TYPE "PLC-Axis"	// UDT 31
VERSION : 0.0
  STRUCT
   A_FD_OR : BYTE ;	//Feedrate override
   A_DriveEnable : BOOL ;	//Drive test movement enable
   A_AckFixedStop : BOOL ;	//Acknowledge fixed stop reached
   A_SensorFixedStop : BOOL ;	//Sensor fixed stop
   A_ASpDisable : BOOL ;	//Axis/spindle disable
   A_Follow_upMode : BOOL ;	//Follow-up mode
   A_PosMeas1 : BOOL ;	//Position measuring system 1
   A_PosMeas2 : BOOL ;	//Position measuring system 2
   A_ORactive : BOOL ;	//Override active
   A_SWCam : BOOL ;	//SW cam activation
   A_ContrEnable : BOOL ;	//Controller enable
   A_DelDTGSpReset : BOOL ;	//Delete distance to go/Spindle-Reset
   A_Clamp : BOOL ;	//Clamping in progress
   A_RefVal1 : BOOL ;	//Reference point value 1
   A_RefVal2 : BOOL ;	//Reference point value 2
   A_RefVal3 : BOOL ;	//Reference point value 3
   A_RefVal4 : BOOL ;	//Reference point value 4
   A_ExtZO : BOOL ;	//Import external ZO
   A_EnabTravFixedStop : BOOL ;	//Enable travel to fixed stop
   A_FixedFD1 : BOOL ;	//Activate fixed feed 1
   A_FixedFD2 : BOOL ;	//Activate fixed feed 2
   A_FixedFD3 : BOOL ;	//Activate fixed feed 3
   A_FixedFD4 : BOOL ;	//Activate fixed feed 4
   A_VelocSpeedLimit : BOOL ;	//Velocity/spindle speed limitation
   A_PrgtestAxRel : BOOL ;	// Program test axis/spindle release
   A_HW1 : BOOL ;	//Activate handwheel 1
   A_HW2 : BOOL ;	//Activate handwheel 2
   A_HW3 : BOOL ;	//Activate handwheel 3
   A_FDSpStop : BOOL ;	//Feed stop/spindle stop
   A_Disable : BOOL ;	//Traversing key disable
   A_RapidTrOR : BOOL ;	//Rapid traverse override
   A_Minus : BOOL ;	//Traversing key minus
   A_Plus : BOOL ;	//Traversing key plus
   A_INC1 : BOOL ;	//INC1
   A_INC10 : BOOL ;	//INC10
   A_INC100 : BOOL ;	//INC100
   A_INC1000 : BOOL ;	//INC1000
   A_INC10000 : BOOL ;	//INC10000
   A_INCVar : BOOL ;	//INC variable
   A_OEMAxis : BYTE ;	//OEM axis signals
   A_InvHWDirOfRot : BOOL ;	// Inverting handwheel direction of rotation
   f7_1 : BOOL ;
   f7_2 : BOOL ;
   f7_3 : BOOL ;
   f7_4 : BOOL ;
   f7_5 : BOOL ;
   f7_6 : BOOL ;
   f7_7 : BOOL ;
   A_NCASpChanA : BOOL ;	//Assign NC axis/spindle channel A
   A_NCASpChanB : BOOL ;	//Assign NC axis/spindle channel B
   A_NCASpChanC : BOOL ;	//Assign NC axis/spindle channel C
   A_NCASpChanD : BOOL ;	//Assign NC axis/spindle channel D
   A_NCASpStrobe : BOOL ;	//Activation of assignment with pos. edge
   f8_5 : BOOL ;
   f8_6 : BOOL ;
   A_PLCASp : BOOL ;	//Request PLC axis/spindle
   A_Para_A : BOOL ;	//Parameter block servo A
   A_Para_B : BOOL ;	//Parameter block servo B
   A_Para_C : BOOL ;	//Parameter block servo C
   A_LockParSetDef : BOOL ;	//Lock parameter set definition from NC
   f9_4 : BOOL ;
   f9_5 : BOOL ;
   f9_6 : BOOL ;
   f9_7 : BOOL ;
   A_REPOSDelay : BOOL ;	//REPOS DELAY
   f10_1 : BOOL ;
   f10_2 : BOOL ;
   f10_3 : BOOL ;
   f10_4 : BOOL ;
   f10_5 : BOOL ;
   f10_6 : BOOL ;
   f10_7 : BOOL ;
   A_StartBrakeTest : BOOL ;	// Start brake test
   f11_1 : BOOL ;
   f11_2 : BOOL ;
   f11_3 : BOOL ;
   f11_4 : BOOL ;
   f11_5 : BOOL ;
   f11_6 : BOOL ;
   f11_7 : BOOL ;
   A_HWLimitMinus : BOOL ;	//Hardware limit switch minus
   A_HWLimitPlus : BOOL ;	//Hardware limit switch plus
   A_SWLimit2Minus : BOOL ;	//2nd software limit switch minus
   A_SWLimit2Plus : BOOL ;	//2nd software limit switch plus
   A_ModuloLimitEn : BOOL ;	// Modulo limit enabled
   f12_5 : BOOL ;
   f12_6 : BOOL ;
   A_DelayRef : BOOL ;	//Delay reference point approach
   A_JogFixPPos0 : BOOL ;	// JogFixPointPos 0
   A_JogFixPPos1 : BOOL ;	// JogFixPointPos 1
   A_JogFixPPos2 : BOOL ;	// JogFixPointPos 2
   A_JogToPos : BOOL ;	// Jog to position
   f13_4 : BOOL ;
   f13_5 : BOOL ;
   f13_6 : BOOL ;
   f13_7 : BOOL ;
   A_ProgtestSuppress : BOOL ;	// Program test to supress
   A_ProgtestActivate : BOOL ;	// Program test activate
   f14_2 : BOOL ;
   f14_3 : BOOL ;
   f14_4 : BOOL ;
   f14_5 : BOOL ;
   f14_6 : BOOL ;
   f14_7 : BOOL ;
   f15 : BYTE ;
   A_ActGearA : BOOL ;	//Actual gear stage A
   A_ActGearB : BOOL ;	//Actual gear stage B
   A_ActGearC : BOOL ;	//Actual gear stage C
   A_GearChangeOv : BOOL ;	//Gear has changed over
   A_Sp1Syn : BOOL ;	//Re-synchronize spindle 1
   A_Sp2Syn : BOOL ;	//Re-synchronize spindle 2
   A_NoMonitorGear : BOOL ;	//No monitoring when changing gear
   A_DeleteS : BOOL ;	//Delete S value
   A_FD_ORSp : BOOL ;	//Feedrate override for spindle valid
   f17_1 : BOOL ;
   f17_2 : BOOL ;
   f17_3 : BOOL ;
   A_Sp1SynP : BOOL ;	//Re-synchronize spindle 1 f. positioning
   A_Sp2SynP : BOOL ;	//Re-synchronize spindle 2 f. positioning
   A_M3M4Inv : BOOL ;	//Invert M3/M4
   f17_7 : BOOL ;
   f18_0 : BOOL ;
   f18_1 : BOOL ;
   f18_2 : BOOL ;
   f18_3 : BOOL ;
   A_OscilPLC : BOOL ;	//Oscillation via PLC
   A_OscilSpeed : BOOL ;	//enable Oscillation
   A_SetRotDirectRight : BOOL ;	//Setpoint osci. direct. right
   A_SetRotDirectLeft : BOOL ;	//Setpoint osci. direct. left
   A_SpOR : BYTE ;	//Spindle override
   f20_0 : BOOL ;
   A_RUEncQuStop : BOOL ;	//Run-up encoder quick stop
   f20_2 : BOOL ;
   A_SpeedSetpSmooth : BOOL ;	//Speed setpoint smoothing
   f20_4 : BOOL ;
   A_HoldBrakeToOpen : BOOL ;	// holding brake open
   f20_6 : BOOL ;
   f20_7 : BOOL ;
   A_ParA : BOOL ;	//Parameter set selection A
   A_ParB : BOOL ;	//Parameter set selection B
   A_ParC : BOOL ;	//Parameter set selection C
   A_MotA : BOOL ;	//Motor selection A
   A_MotB : BOOL ;	//Motor selection B
   A_MotOK : BOOL ;	//Motor selected
   A_IntegratDisable : BOOL ;	//n controller integrator disable
   A_PulseEnable : BOOL ;	//Pulse enable
   A_SG_SBH : BOOL ;	//Deselection SG/SBH
   A_SBH : BOOL ;	//Deselection of safe standstill
   f22_2 : BOOL ;
   A_SGselect0 : BOOL ;	//Selection SG bit 0
   A_SGselect1 : BOOL ;	//Selection SG bit 1
   f22_5 : BOOL ;
   f22_6 : BOOL ;
   f22_7 : BOOL ;
   A_Transmiss0 : BOOL ;	//Selection Transmission bit 0
   A_Transmiss1 : BOOL ;	//Selection Transmission bit 1
   A_Transmiss2 : BOOL ;	//Selection Transmission bit 2
   f23_3 : BOOL ;
   A_SE : BOOL ;	//Selection SE
   A_BrakeToClose : BOOL ;	//Sinamics: Brake to close
   f23_6 : BOOL ;
   A_TestStop : BOOL ;	//Activate test stop
   A_RotationMonit : BOOL ;	// Stepper motor: Rotation monitoring
   A_ControlAx : BOOL ;	// Control Axis
   f24_2 : BOOL ;
   f24_3 : BOOL ;
   A_TorqComp : BOOL ;	// Torque compensation
   A_ChangSetpOutAss0 : BOOL ;	// Bit value for CTRLOUT_changed - Change setpoint output assignment
   A_ChangSetpOutAss1 : BOOL ;	// Bit value for CTRLOUT_changed - Change setpoint output assignment
   A_MS : BOOL ;	//Master / Slave On
   f25 : BYTE ;
   f26_0 : BOOL ;
   f26_1 : BOOL ;
   f26_2 : BOOL ;
   A_CompContr : BOOL ;	//Compensation controller On
   A_FollowAxOv : BOOL ;	//Enable following axis override
   f26_5 : BOOL ;
   f26_6 : BOOL ;
   f26_7 : BOOL ;
   A_DEPMCS : BOOL ;	// Resume: DEPMCS
   A_DEPBCS : BOOL ;	// Resume: DEPBCS
   A_Corr : BOOL ;	// Resume: Corr
   A_HIAxMove : BOOL ;	// Resume: HIAxMove
   A_StopDEPMCS : BOOL ;	// Stop: DEPMCS
   A_StopDEPBCS : BOOL ;	// Stop: DEPBCS
   A_StopCorr : BOOL ;	// Stop: Corr
   A_StopHIAxMove : BOOL ;	// Stop: HIAxMove
   A_OscillAxExtRev : BOOL ;	// OscillAxExtReversal
   A_AxReset : BOOL ;	// AXRESET
   A_AxResume : BOOL ;	// AXRESUME
   A_SetRP : BOOL ;	//Set reversal point
   A_ChangeRP : BOOL ;	//Change reversal point
   A_StopRP : BOOL ;	//Stop at next reversal point
   A_Stop : BOOL ;	//Stop
   A_PLCAxis : BOOL ;	//PLC checks axis
   f29_0 : BOOL ;
   f29_1 : BOOL ;
   f29_2 : BOOL ;
   f29_3 : BOOL ;
   A_StartGantSynRun : BOOL ;	//Start gantry synchronization run
   A_NoAutoSync : BOOL ;	//No auto sync
   f29_6 : BOOL ;
   f29_7 : BOOL ;
   A_StopSpindle : BOOL ;	//Stop spindle
   A_StartCW : BOOL ;	//Start spindle Clockwise
   A_StartCCW : BOOL ;	//Start spindle Counterclockwise
   A_AutoGearStep : BOOL ;	//Autom. gear step change
   A_PosSpindle : BOOL ;	//Position spindle
   f30_5 : BOOL ;
   f30_6 : BOOL ;
   f30_7 : BOOL ;
   f31_0 : BOOL ;
   f31_1 : BOOL ;
   f31_2 : BOOL ;
   f31_3 : BOOL ;
   A_Resynchronize : BOOL ;	// Resynchronize
   A_DisSync : BOOL ;	// Disable synchronization
   A_Tracksync : BOOL ;	// Track synchronism
   A_DelSyncRunCorr : BOOL ;	// Deleting synchronous run correction
   f32_0 : BOOL ;
   f32_1 : BOOL ;
   A_extStopA : BOOL ;	//Deselection external Stop A
   A_extStopC : BOOL ;	//Deselection external Stop C
   A_extStopD : BOOL ;	//Deselection external Stop D
   A_extStopE : BOOL ;	//Deselection external Stop E
   f32_6 : BOOL ;
   f32_7 : BOOL ;
   f33_0 : BOOL ;
   f33_1 : BOOL ;
   f33_2 : BOOL ;
   f33_3 : BOOL ;
   A_SGcorr_0 : BOOL ;	//Selection SG-correction Bit 0
   A_SGcorr_1 : BOOL ;	//Selection SG-correction Bit 1
   A_SGcorr_2 : BOOL ;	//Selection SG-correction Bit 2
   A_SGcorr_3 : BOOL ;	//Selection SG-correction Bit 3
   f34 : ARRAY  [34 .. 55 ] OF BYTE ;
   A_FeedDriveCAxEng : BOOL ;	// Seperate feed drive as C axis engaged
   A_SpSpeedDisp : BOOL ;	// Spindle speed display
   A_SpInsideClamp : BOOL ;	// Spindle inside clamping
   f56_3 : BOOL ;
   f56_4 : BOOL ;
   f56_5 : BOOL ;
   f56_6 : BOOL ;
   f56_7 : BOOL ;
   f57 : BYTE ;
   f58 : WORD ;	// FC18: internal
   E_SpNA : BOOL ;	//Spindle/no axis
   E_NCU_Link : BOOL ;	//NCU_link active axis
   E_EncodFreq1 : BOOL ;	//Encoder limit frequency 1 exceeded
   E_EncodFreq2 : BOOL ;	//Encoder limit frequency 2 exceeded
   E_RefSyn1 : BOOL ;	//Referenced/synchronized 1
   E_RefSyn2 : BOOL ;	//Referenced/synchronized 2
   E_ExactCoarse : BOOL ;	//Position reached with exact stop coarse
   E_ExactFine : BOOL ;	//Position reached with exact stop fine
   E_TravRequ : BOOL ;	//Travel request
   E_AxialAlarm : BOOL ;	// Axial alarm
   E_AxisReady : BOOL ;	//Axis ready
   E_Follow_upMode : BOOL ;	//Follow-up mode active
   E_Stat : BOOL ;	//Axis/spindle stationary (n<nmin)
   E_PositContr : BOOL ;	//Position controller active
   E_SpeedContr : BOOL ;	//Speed controller active
   E_CurrentContr : BOOL ;	//Current controller active
   E_SWCam : BOOL ;	//Software cams active
   E_HWOverlay : BOOL ;	//Handwheel overlay active
   E_RevFD : BOOL ;	//Revolutional feedrate active
   E_MeasAct : BOOL ;	//Measuring active
   E_ActTravFStop : BOOL ;	//Activate travel to fixed stop
   E_FixedStop : BOOL ;	//Fixed stop reached
   E_ForceFixedStop : BOOL ;	// Force fixed stop limited
   E_AxContainerRot : BOOL ;	// Axis container rotation active
   E_AxReset : BOOL ;	// Axis reset done
   E_PLCCtrlAx : BOOL ;	// PLCcontrolled axis
   E_AxStop : BOOL ;	// Axis stop active
   E_AxSpDisable : BOOL ;	// Axis/spindle disable active
   E_StopDEPMCS : BOOL ;	// stop DEPMCS active
   E_StopDEPBCS : BOOL ;	// stop DEPBCS active
   E_StopCorr : BOOL ;	// stop Corr active
   E_StopHIAxMove : BOOL ;	// Stop HIAxMove active
   E_HW1 : BOOL ;	//Handwheel 1 active
   E_HW2 : BOOL ;	//Handwheel 2 active
   E_HW3 : BOOL ;	//Handwheel 3 active
   f64_3 : BOOL ;
   E_TReqMinus : BOOL ;	// Travel request minus
   E_TReqPlus : BOOL ;	// Travel request plus
   E_TCMinus : BOOL ;	//Traverse command minus
   E_TCPlus : BOOL ;	//Traverse command plus
   E_INC1 : BOOL ;	//INC1
   E_INC10 : BOOL ;	//INC10
   E_INC100 : BOOL ;	//INC100
   E_INC1000 : BOOL ;	//INC1000
   E_INC10000 : BOOL ;	//INC10000
   E_INCVar : BOOL ;	//INC variable
   f65_6 : BOOL ;
   f65_7 : BOOL ;
   E_OEMAxis : BYTE ;	//OEM axis signals
   E_InvHWDirOfRot : BOOL ;	// Handwheel direction of rotation invert actively
   f67_1 : BOOL ;
   f67_2 : BOOL ;
   f67_3 : BOOL ;
   f67_4 : BOOL ;
   f67_5 : BOOL ;
   f67_6 : BOOL ;
   f67_7 : BOOL ;
   E_NCASpChanA : BOOL ;	//NC axis/spindle in channel A
   E_NCASpChanB : BOOL ;	//NC axis/spindle in channel B
   E_NCASpChanC : BOOL ;	//NC axis/spindle in channel C
   E_NCASpChanD : BOOL ;	//NC axis/spindle in channel D
   E_PLCType : BOOL ;	//New type requested by PLC
   E_ChPoss : BOOL ;	//Change axis possible
   E_NeutrASp : BOOL ;	//Neutral axis/spindle
   E_PLCASp : BOOL ;	//PLC axis/spindle
   E_ParS_A : BOOL ;	//Parameter block servo A
   E_ParS_B : BOOL ;	//Parameter block servo B
   E_ParS_C : BOOL ;	//Parameter block servo C
   E_NCUNumLink_3 : BOOL ;
   E_NCUNumLink_4 : BOOL ;
   E_NCUNumLink_5 : BOOL ;
   E_NCUNumLink_6 : BOOL ;
   E_NCUNumLink_7 : BOOL ;
   E_ReposSh : BOOL ;	// Repos shift
   E_ReposShValid : BOOL ;	// Repos shift valid
   E_ReposDelayQuit : BOOL ;	// Repos delay quit
   f70_3 : BOOL ;
   f70_4 : BOOL ;
   f70_5 : BOOL ;
   f70_6 : BOOL ;
   f70_7 : BOOL ;
   E_BrakeTest : BOOL ;	// Brake test active
   f71_1 : BOOL ;
   f71_2 : BOOL ;
   f71_3 : BOOL ;
   E_POS_RESTORED1 : BOOL ;	// POS_RESTORED 1
   E_POS_RESTORED2 : BOOL ;	// POS_RESTORED 2
   f71_6 : BOOL ;
   E_PLCAxDedic : BOOL ;	// PLC Axis dedicated
   E_MMC_REPOSDelay : BOOL ;	//MMC REPOS DELAY
   f72_1 : BOOL ;
   f72_2 : BOOL ;
   f72_3 : BOOL ;
   f72_4 : BOOL ;
   f72_5 : BOOL ;
   f72_6 : BOOL ;
   f72_7 : BOOL ;
   f73 : BYTE ;
   f74_0 : BOOL ;
   f74_1 : BOOL ;
   f74_2 : BOOL ;
   f74_3 : BOOL ;
   E_ModLimEnAct : BOOL ;	// Modulo limit enabled active
   f74_5 : BOOL ;
   f74_6 : BOOL ;
   f74_7 : BOOL ;
   E_JogFixPPos0Act : BOOL ;	// JogFixPointPos 0 active
   E_JogFixPPos1Act : BOOL ;	// JogFixPointPos 1 active
   E_JogFixPPos2Act : BOOL ;	// JogFixPointPos 2 active
   E_JogFixPPos0 : BOOL ;	// JogFixPointPos 0 reached
   E_JogFixPPos1 : BOOL ;	// JogFixPointPos 1 reached
   E_JogFixPPos2 : BOOL ;	// JogFixPointPos 2 reached
   E_JogToPos : BOOL ;	// Jog to position active
   E_JogPos : BOOL ;	// Jog position reached
   E_ScratchPulse : BOOL ;	//Scratch pulse
   f76_1 : BOOL ;
   f76_2 : BOOL ;
   f76_3 : BOOL ;
   E_PathAxis : BOOL ;	// Path axis
   E_PosAxis : BOOL ;	//Positioning axis
   E_IndexAxisPos : BOOL ;	//Indexing axis in position
   E_CurvePos : BOOL ;	//Curve axis in position
   E_CollCheckRedSpeed : BOOL ;	//reduced speed of Collisions Check
   f77_1 : BOOL ;
   f77_2 : BOOL ;
   f77_3 : BOOL ;
   f77_4 : BOOL ;
   f77_5 : BOOL ;
   f77_6 : BOOL ;
   f77_7 : BOOL ;
   E_FPosAxis : REAL ;	//F function (REAL format) for positioning axes
   E_SetpGearA : BOOL ;	//Setpoint gear stage A
   E_SetpGearB : BOOL ;	//Setpoint gear stage B
   E_SetpGearC : BOOL ;	//Setpoint gear stage C
   E_GearChange : BOOL ;	//Gear changeover
   f82_4 : BOOL ;
   f82_5 : BOOL ;
   f82_6 : BOOL ;
   f82_7 : BOOL ;
   E_SpeedLimit : BOOL ;	//Speed limit exceeded
   E_SetSpeedLimit : BOOL ;	//Setpoint speed limited
   E_SetSpeedIncreased : BOOL ;	//Setpoint speed increased
   E_GeoMonit : BOOL ;	//Geometry monitoring
   E_SupportAreaViol : BOOL ;	//Support area limits violated
   E_SetRange : BOOL ;	//Spindle in setpoint range
   E_SpeedMonit : BOOL ;	//Speed monitoring
   E_ActRotRight : BOOL ;	//Actual rotation direction right
   E_ConstCuttSpeed : BOOL ;	//Const. cutting speed active
   E_SUG : BOOL ;	//SUG active (grinding wheel surface speed)
   E_CLG : BOOL ;	//CLG active
   E_Tapping : BOOL ;	//Tapping without compensating chuck
   E_SyncMode : BOOL ;	//Synchronous mode spindle active
   E_PosMode : BOOL ;	//Positioning mode spindle active
   E_OscillMode : BOOL ;	//Oscillation mode spindle active
   E_ContrMode : BOOL ;	//Control mode spindle active
   E_ToolDynLimit : BOOL ;	// Tool with limit of dynamics
   f85_1 : BOOL ;
   f85_2 : BOOL ;
   f85_3 : BOOL ;
   f85_4 : BOOL ;
   E_SpInPosition : BOOL ;	// Spindle in position
   f85_6 : BOOL ;
   f85_7 : BOOL ;
   E_MFunct : INT ;	//M function (INT) for spindle
   E_SFunct : REAL ;	//S function (REAL) for spindle
   f92_0 : BOOL ;
   E_RUEncDisabl : BOOL ;	//Run-up encoder disable active
   f92_2 : BOOL ;
   E_SpeedSetpSmooth : BOOL ;	//Speed setpoint smoothing active
   E_RLIact : BOOL ;	// RLI active
   E_HoldBrakeOpened : BOOL ;	// Holding brake opened
   f92_6 : BOOL ;
   f92_7 : BOOL ;
   E_ParA : BOOL ;	//Active parameter set A
   E_ParB : BOOL ;	//Active parameter set B
   E_ParC : BOOL ;	//Active parameter set C
   E_MotA : BOOL ;	//Active motor A
   E_MotB : BOOL ;	//Active motor B
   E_MotOK : BOOL ;	//Drive ready
   E_IntegratDisable : BOOL ;	//n controller integrator disabled
   E_PulseEnable : BOOL ;	//Pulses enabled
   E_MTempWarn : BOOL ;	//Temperature prewarning motor
   E_HTempWarn : BOOL ;	//Temperature prewarning heat sink
   E_RUComplete : BOOL ;	//Ramp-up complete
   E_MdMdx : BOOL ;	//Md<Mdx
   E_NactNmin : BOOL ;	//nact<nmin
   E_NactNx : BOOL ;	//nact<nx
   E_NactNset : BOOL ;	//nact<nset
   E_Message : BOOL ;	//Variable message function
   E_UDClessAlThreshold : BOOL ;	//UDC-link < alarm threshold
   f95_1 : BOOL ;
   f95_2 : BOOL ;
   f95_3 : BOOL ;
   f95_4 : BOOL ;
   f95_5 : BOOL ;
   f95_6 : BOOL ;
   f95_7 : BOOL ;	// Power Section I2T limit
   E_SpindleMonit : BOOL ;	//Error spindle monitoring
   E_AxisCtrl : BOOL ;	// Axis control active
   E_MSFine : BOOL ;	// Master/Slave fine
   E_MSCoarse : BOOL ;	// Master/Slave coarse
   E_MSCompContr : BOOL ;	// Master/Slave Compensation controller activ
   E_BitValCtrlOutChang0 : BOOL ;	// Bit value for CTRLOUT_changed 0:  Change setpoint output assignment
   E_BitValCtrlOutChang1 : BOOL ;	// Bit value for CTRLOUT_changed 1:  Change setpoint output assignment
   E_MS : BOOL ;	//Master/ slave active
   f97 : BYTE ;
   E_SyncronFine : BOOL ;	//Synchronism fine
   E_SyncronCoarse : BOOL ;	//Synchronism coarse
   E_ActValCoupling : BOOL ;	//Actual value coupling
   f98_3 : BOOL ;
   E_OverlayMotion : BOOL ;	//Overlaid motion
   E_SWL : BOOL ;	//Speed warning limit reached
   E_AWL : BOOL ;	//Acceleration warning limit reached
   E_EmRetr : BOOL ;	//Emergency retraction active
   E_MasterSp : BOOL ;	//Master spindle
   E_SlaveSp : BOOL ;	//Slave spindle
   E_SyncRunCorrDOut : BOOL ;	// Synchronous run correction driven out
   E_AxisAccel : BOOL ;	//Axis accelerated
   E_Sync : BOOL ;	//Synchronization active
   E_MSR : BOOL ;	//Max speed reached
   E_MAR : BOOL ;	//Max acceleration reached
   f99_7 : BOOL ;
   f100_0 : BOOL ;
   f100_1 : BOOL ;
   E_OscillAxExtRev : BOOL ;	// OscillAxExt Reversal active
   E_StopOscill : BOOL ;	//Oscillation cannot start
   E_ErrorOscill : BOOL ;	//Error during oscillation
   E_SparkOut : BOOL ;	//Spark-out active
   E_OscillMotion : BOOL ;	//Oscillation motion active
   E_Oscill : BOOL ;	//Oscillation active
   f101_0 : BOOL ;
   f101_1 : BOOL ;
   E_GantCOLimit : BOOL ;	//Gantry cut-off limit exceeded
   E_GantWarn : BOOL ;	//Gantry warning limit exceeded
   E_SynRunStart : BOOL ;	//Synchronization run ready to start
   E_GantGroupSyn : BOOL ;	//Gantry grouping is synchronous
   E_GantLeadAxis : BOOL ;	//Gantry leading axis
   E_GantAxis : BOOL ;	//Gantry axis
   f102 : BYTE ;
   E_SyncRunCorrIncl : BOOL ;	// Synchronous run correction is included
   f103_1 : BOOL ;
   f103_2 : BOOL ;
   f103_3 : BOOL ;
   f103_4 : BOOL ;
   f103_5 : BOOL ;
   f103_6 : BOOL ;
   f103_7 : BOOL ;
   E_AIAxis : ARRAY  [1 .. 31 ] OF BOOL ;	//Active infeed axis[1..31]
   E_SG_SBH : BOOL ;	//Active SG/SBH
   E_ErrLifeS_CRC : BOOL ;	// Error lifesign or CRC-error
   E_ImpdelNCK : BOOL ;	//Delete pulses NCK
   r108_3 : BOOL ;
   r108_4 : BOOL ;
   r108_5 : BOOL ;
   r108_6 : BOOL ;
   E_SRef : BOOL ;	//Axis safely referenced
   E_SN1Plus : BOOL ;	//Actual position > cam position SN1+
   E_SN1Minus : BOOL ;	//Actual position > cam position SN1-
   E_SN2Plus : BOOL ;	//Actual position > cam position SN2+
   E_SN2Minus : BOOL ;	//Actual position > cam position SN2-
   E_SN3Plus : BOOL ;	//Actual position > cam position SN3+
   E_SN3Minus : BOOL ;	//Actual position > cam position SN3-
   E_SN4Plus : BOOL ;	//Actual position > cam position SN4+
   E_SN4Minus : BOOL ;	//Actual position > cam position SN4-
   f110_0 : BOOL ;
   E_SBH : BOOL ;	//Active SBH
   f110_2 : BOOL ;
   E_SG_0 : BOOL ;	//Active SG 0
   E_SG_1 : BOOL ;	//Active SG 1
   E_n_nx : BOOL ;	//n < nx
   f110_6 : BOOL ;
   f110_7 : BOOL ;
   f111_0 : BOOL ;
   f111_1 : BOOL ;
   f111_2 : BOOL ;
   f111_3 : BOOL ;
   E_StopAB : BOOL ;	//Stop A/B active
   E_StopC : BOOL ;	//Stop C active
   E_StopD : BOOL ;	//Stop D active
   E_StopE : BOOL ;	//Stop E active
   E_CamRangeTr1 : BYTE ;	//Cam Range for Cam Track 1
   E_CamRangeTr2 : BYTE ;	//Cam Range for Cam Track 2
   E_CamRangeTr3 : BYTE ;	//Cam Range for Cam Track 3
   E_CamRangeTr4 : BYTE ;	//Cam Range for Cam Track 4
   f116 : BYTE ;
   E_CamTrack1 : BOOL ;	//Cam Track 1
   E_CamTrack2 : BOOL ;	//Cam Track 2
   E_CamTrack3 : BOOL ;	//Cam Track 3
   E_CamTrack4 : BOOL ;	//Cam Track 4
   f117_4 : BOOL ;
   f117_5 : BOOL ;
   f117_6 : BOOL ;
   f117_7 : BOOL ;
   E_CamRangeBitTr1 : ARRAY  [0 .. 14 ] OF //Cam Range Bits for Cam Track 1
   BOOL ;
   E_CamRangeBitTr2 : ARRAY  [0 .. 14 ] OF //Cam Range Bits for Cam Track 2
   BOOL ;
   E_CamRangeBitTr3 : ARRAY  [0 .. 14 ] OF //Cam Range Bits for Cam Track 3
   BOOL ;
   E_CamRangeBitTr4 : ARRAY  [0 .. 14 ] OF //Cam Range Bits for Cam Track 4
   BOOL ;
   f126 : WORD ;	// internal
   E_MMC_ProgtestSuppress : BOOL ;	// HMI->PLC: Program test to supress
   E_MMC_ProgtestActivate : BOOL ;	// HMI->PLC: Program test activate
   f128_2 : BOOL ;
   f128_3 : BOOL ;
   f128_4 : BOOL ;
   f128_5 : BOOL ;
   f128_6 : BOOL ;
   f128_7 : BOOL ;
   f129 : BYTE ;
   f130 : WORD ;
   E_SensorAv : BOOL ;	// Sensors available
   E_S1aMeasARod : BOOL ;	// Sensor S1: analogous measurement position of actuating rod
   f132_2 : BOOL ;
   f132_3 : BOOL ;
   E_S4dPistonStopP : BOOL ;	// Sensor S4: digital value piston stop position
   E_S5dAngleShaft : BOOL ;	// Sensor S5: digital value angle situation shaft
   f132_6 : BOOL ;
   f132_7 : BOOL ;
   f133 : BYTE ;
   E_ClampingState : INT ;	// state of the clamping system
   E_AnalogSensor : INT ;	// analog sensor on the motor
   f138_0 : BOOL ;
   f138_1 : BOOL ;
   f138_2 : BOOL ;
   f138_3 : BOOL ;
   E_S4PistonStopP : BOOL ;	// Sensor S4: piston stop position
   E_S5AngleShaft : BOOL ;	// Sensor S5: angle situation shaft
   f138_6 : BOOL ;
   f138_7 : BOOL ;
   f139 : BYTE ;
  END_STRUCT ;	
END_TYPE

// UDT 62: know-how protected block, not included

TYPE UDT 71
VERSION : 0.0
  STRUCT
   IFNo : ARRAY  [1 .. 16 ] OF BOOL ;	//Interface [no.] active
   Quit : ARRAY  [1 .. 16 ] OF BOOL ;	//perform Quit-End
   IF : ARRAY  [1 .. 16 ] OF STRUCT
    Loading : BOOL ;
    Unloading : BOOL ;
    Reloading : BOOL ;
    Positioning : BOOL ;
    PosbyProgram : BOOL ;	//Initiation by CNC Program
    PositioningMT : BOOL ;	//Positioning Multitool
    f0_6 : BOOL ;
    f0_7 : BOOL ;
    PerfStatusError : BOOL ;
    n1_1 : BOOL ;
    n1_2 : BOOL ;
    n1_3 : BOOL ;
    n1_4 : BOOL ;
    n1_5 : BOOL ;
    n1_6 : BOOL ;
    DataInDB1071 : BOOL ;
    Channel : BYTE ;	//Assigned channel
    TMno : BYTE ;	//Tool management no.
    Free1 : DINT ;	//Unassigned parameter 1
    Free2 : DINT ;	//Unassigned parameter 2
    Free3 : DINT ;	//Unassigned parameter 3
    IdentLoad : INT ;	//Identification for loading/unloading station
    NoLoad : INT ;	//No. of loading station
    SMag : INT ;	//Magazine no. (source) for unloading/reloading/pos.
    SLoc : INT ;	//Location no. (source) for unloading/reloading/pos.
    TMag : INT ;	//Magazine no. (target) for loading/reloading
    TLoc : INT ;	//Location no. (target) for loading/reloading
    WithoutMagMoving : BOOL ;	//HMI Data: Without Magazine Moving
    Res2 : BYTE ;
   END_STRUCT ;
  END_STRUCT ;	
END_TYPE

TYPE UDT 72
VERSION : 0.0
  STRUCT
   IFNo : ARRAY  [1 .. 16 ] OF BOOL ;	//Interface [no.] active
   Quit : ARRAY  [1 .. 16 ] OF BOOL ;	//perform Quit-End
   IF : ARRAY  [1 .. 16 ] OF STRUCT
    Comp : BOOL ;	//Compulsory change
    Perform : BOOL ;	//Perform change
    Prepare : BOOL ;	//Prepare change
    T0 : BOOL ;	//T0 programmed
    OldTinDBW42 : BOOL ;	//ZWS No. of Old Tool in DBW (n+42)
    ManTIn : BOOL ;	//Put in Tool in Spindle manual
    ManTOut : BOOL ;	//Get out Tool from Spindle manual
    SpiTRSpi : BOOL ;	//Spindle Tool remains in spindle
    PerfStatusError : BOOL ;
    n1_1 : BOOL ;
    n1_2 : BOOL ;
    n1_3 : BOOL ;
    n1_4 : BOOL ;
    n1_5 : BOOL ;
    n1_6 : BOOL ;
    DataInDB1072 : BOOL ;
    Channel : BYTE ;	//Assigned channel
    TMno : BYTE ;	//Tool management no.
    Free1 : DINT ;	//Unassigned parameter 1
    Free2 : DINT ;	//Unassigned parameter 2
    Free3 : DINT ;	//Unassigned parameter 3
    IdentBuff : INT ;	//Buffer identification (fixed value 9998)
    NoBuff : INT ;	//Relative location (target) in the buffer
    SMag : INT ;	//Magazine no. (source) for new tool
    SLoc : INT ;	//Location no. (source) for new tool
    TMag : INT ;	//Magazine no. (target) for old tool
    TLoc : INT ;	//Location no. (target) for old tool
    LocType : INT ;	//Tool new: location type
    SLeft : INT ;	//Tool new: size left
    SRight : INT ;	//Tool new: size right
    STop : INT ;	//Tool new: size top
    SBottom : INT ;	//Tool new: size bottom
    ToolInBuff : BOOL ;	//ID for tools in buffer
    IgnoreDisab : BOOL ;	//Ignore disabled
    TBUnloaded : BOOL ;	//To be unloaded
    TBLoaded : BOOL ;	//To be loaded
    MasterTool : BOOL ;	//Master tool
    n38_5 : BOOL ;	//reserved
    Exchange_1to1 : BOOL ;	//1:1 exchange
    HandTool : BOOL ;	//Hand tool
    ActTool : BOOL ;	//Active tool
    ToolEnabl : BOOL ;	//Tool enabled
    ToolDisab : BOOL ;	//Tool disabled
    Measured : BOOL ;	//Tool measured
    Prewarn : BOOL ;	//Prewarning limit reached
    ToolChange : BOOL ;	//Tool being changed
    FixedLoc : BOOL ;	//Tool fixed location coded
    ToolUsed : BOOL ;	//Tool was in use
    T_no : INT ;	//Tool new: T no.
    OldTZWSNo : INT ;	//ZWS No. of Old Tool
    MyMag : INT ;
    MyPlace : INT ;
   END_STRUCT ;
  END_STRUCT ;	
END_TYPE

TYPE UDT 73
VERSION : 0.0
  STRUCT
   IfNo : ARRAY  [1 .. 16 ] OF BOOL ;	//Interface [no.] active
   Quit : ARRAY  [1 .. 16 ] OF BOOL ;	//perform Quit-End
   IF : ARRAY  [1 .. 16 ] OF STRUCT
    Comp : BOOL ;	//Compulsory change
    Perform : BOOL ;	//Perform change
    f0_2 : BOOL ;
    T0 : BOOL ;	//T0 programmed
    f0_4 : BOOL ;
    f0_5 : BOOL ;
    ManTOut : BOOL ;	//Get out Tool from Holder manual
    f0_7 : BOOL ;
    PerfStatusError : BOOL ;
    n1_1 : BOOL ;
    n1_2 : BOOL ;
    n1_3 : BOOL ;
    n1_4 : BOOL ;
    n1_5 : BOOL ;
    n1_6 : BOOL ;
    DataInDB1073 : BOOL ;
    Channel : BYTE ;	//Assigned channel
    TMno : BYTE ;	//Tool management no.
    Free1 : DINT ;	//Unassigned parameter 1
    Free2 : DINT ;	//Unassigned parameter 2
    Free3 : DINT ;	//Unassigned parameter 3
    KennZWS : INT ;	//Reserved (buffer identification)
    NoBuff : INT ;	//Rel. location in buffer (res.)
    SMag : INT ;	//Magazine no. of turret
    SLoc : INT ;	//Location no. for new tool
    TMag : INT ;	//Magazine no. of turret (res.)
    TLoc : INT ;	//Location no. for old tool
    LocType : INT ;	//Tool new: location type
    SLeft : INT ;	//Tool new: size left
    SRight : INT ;	//Tool new: size right
    STop : INT ;	//Tool new: size top
    SBottom : INT ;	//Tool new: size bottom
    ToolInBuff : BOOL ;	//ID for tools in buffer
    IgnoreDisab : BOOL ;	//Ignore disabled
    TBUnloaded : BOOL ;	//To be unloaded
    TBLoaded : BOOL ;	//To be loaded
    MasterTool : BOOL ;	//Master tool
    n38_5 : BOOL ;	//reserved
    Exchange_1to1 : BOOL ;	//1:1 exchange
    HandTool : BOOL ;	//Hand tool
    ActTool : BOOL ;	//Active tool
    ToolEnabl : BOOL ;	//Tool enabled
    ToolDisab : BOOL ;	//Tool disabled
    Measured : BOOL ;	//Tool measured
    Prewarn : BOOL ;	//Prewarning limit reached
    ToolChange : BOOL ;	//Tool being changed
    FixedLoc : BOOL ;	//Tool fixed location coded
    ToolUsed : BOOL ;	//Tool was in use
    T_no : INT ;	//Tool new: T no.
    MyPlace : INT ;
   END_STRUCT ;
  END_STRUCT ;	
END_TYPE

TYPE UDT 77
VERSION : 0.0
  STRUCT
   MCP1In : ARRAY  [0 .. 7 ] OF BYTE ;
   MCP1Out : ARRAY  [0 .. 7 ] OF BYTE ;
   MCP1StatSend : DWORD ;
   MCP1StatRec : DWORD ;
   MCP2In : ARRAY  [0 .. 7 ] OF BYTE ;
   MCP2Out : ARRAY  [0 .. 7 ] OF BYTE ;
   MCP2StatSend : DWORD ;
   MCP2StatRec : DWORD ;
   BHGIn : ARRAY  [0 .. 5 ] OF BYTE ;
   Filler : ARRAY  [0 .. 5 ] OF BYTE ;
   BHGOut : ARRAY  [0 .. 19 ] OF BYTE ;
   BHGStatSend : DWORD ;
   BHGStatRec : DWORD ;
  END_STRUCT ;	
END_TYPE

TYPE UDT 1002
VERSION : 0.0
  STRUCT 	//Offset 0
   Chan : ARRAY  [1 .. 10 ] OF STRUCT 	//From Channel 1 to Channel 10
    FDD : ARRAY  [0 .. 15 ] OF //Feed disable
    BOOL ;
    RID : ARRAY  [0 .. 15 ] OF //Read-in disable
    BOOL ;
    NCSD : ARRAY  [0 .. 15 ] OF //NC start disable
    BOOL ;
    FdStop_1 : ARRAY  [0 .. 15 ] OF //Feed stop GEOaxis 1
    BOOL ;
    FdStop_2 : ARRAY  [0 .. 15 ] OF //Feed stop GEOaxis 2
    BOOL ;
    FdStop_3 : ARRAY  [0 .. 15 ] OF //Feed stop GEOaxis 3
    BOOL ;
   END_STRUCT ;	//without Alarmno for Chan (120 Byte)
//Offset 120
   Axis : ARRAY  [1 .. 31 ] OF STRUCT 	//From Axis 1 to Axis 31
    FdStop : ARRAY  [0 .. 15 ] OF //Feed stop axis/spindle 1
    BOOL ;
   END_STRUCT ;	//without Alarmno for Axis (62 Byte)
//Offset 182
   ZInfo0 : ARRAY  [0 .. 63 ] OF WORD ;	//Additional Value for UserAlarms 700000 to 700063
//Offset 310
   ChanA : ARRAY  [1 .. 10 ] OF STRUCT 	//From Channel 1 to Channel 10
    FDD_5C00xx : ARRAY  [0 .. 15 ] OF //Feed disable A.no.51000-510015
    BOOL ;
    FDD_RID_5C01xx : ARRAY  [0 .. 31 ] OF //Feed and read-in disable A.no.510100-510131
    BOOL ;
    RID_5C02xx : ARRAY  [0 .. 31 ] OF //Read-in disable A.no.510200-510231
    BOOL ;
    NCSD_5C03xx : ARRAY  [0 .. 15 ] OF //NC start disable A.no.510300-510315
    BOOL ;
    FdStop_1_5C11xx : ARRAY  [0 .. 15 ] OF //Feed stop GEOaxis 1 A.no.511100-511115
    BOOL ;
    FdStop_2_5C12xx : ARRAY  [0 .. 15 ] OF //Feed stop GEOaxis 2 A.no.511200-511215
    BOOL ;
    FdStop_3_5C13xx : ARRAY  [0 .. 15 ] OF //Feed stop GEOaxis 3 A.no.511300-511315
    BOOL ;
   END_STRUCT ;	//Alarmno for Chan are 5Cxxxx; C is the ChannelNo, except Channel 10. Channel 10
   AxisA : ARRAY  [1 .. 32 ] OF STRUCT 	//From Axis 1 to Axis 31
    AAFdStop60AAxx : ARRAY  [0 .. 15 ] OF //Feed stop axis/spindle
    BOOL ;
   END_STRUCT ;	//Alarmno for Axis are 60AAxx; A is the Axisno.
//Offset 554
   UserA : ARRAY  [0 .. 31 ] OF STRUCT
    A70UUxx : ARRAY  [0 .. 63 ] OF //Alarm 700000-700063 (user area 0)
    BOOL ;
   END_STRUCT ;	//Alarmno for UserAlarms are 7yUUxx; U is the Userarea, y = Db1004.UserDek2No[U]
  END_STRUCT ;	
END_TYPE

TYPE UDT 1071
VERSION : 0.0
  STRUCT
   MTIF : ARRAY  [1 .. 16 ] OF STRUCT
    MtType : INT ;
    MtPlaces : INT ;
    MtDistance : REAL ;
    MtNum : INT ;	// MT-No. to be positioned to
    MtPlaceNum : INT ;	// MT-PlaceNo. ~
    ToolHolder : INT ;	// TH-No as reference for MT-positioning
    IF : ARRAY  [1 .. 3 ] OF STRUCT
     reserved : INT ;	// reserved
    END_STRUCT ;
   END_STRUCT ;
  END_STRUCT ;	
END_TYPE

TYPE UDT 1072
VERSION : 0.0
  STRUCT
   MTIF : ARRAY  [1 .. 16 ] OF STRUCT
    MtType : INT ;
    MtPlaces : INT ;
    MtDistance : REAL ;
    MtNumNew : INT ;	// MT-No. new Tool
    MtPlaceNumNew : INT ;	// MtoolPlaceNum  ~
    MtNumOld : INT ;	// MT-No. old Tool
    MtPlaceNumOld : INT ;	// MtoolPlaceNum  ~
    LocType : INT ;	//Tool new: location type
    SLeft : INT ;	//Tool new: size left
    SRight : INT ;	//Tool new: size right
    STop : INT ;	//Tool new: size top
    SBottom : INT ;	//Tool new: size bottom
    ToolInBuff : BOOL ;	//ID for tools in buffer
    IgnoreDisab : BOOL ;	//Ignore disabled
    TBUnloaded : BOOL ;	//To be unloaded
    TBLoaded : BOOL ;	//To be loaded
    MasterTool : BOOL ;	//Master tool
    n26_5 : BOOL ;	//reserved
    n26_6 : BOOL ;	//reserved
    HandTool : BOOL ;	//Hand tool
    ActTool : BOOL ;	//Active tool
    ToolEnabl : BOOL ;	//Tool enabled
    ToolDisab : BOOL ;	//Tool disabled
    Measured : BOOL ;	//Tool measured
    Prewarn : BOOL ;	//Prewarning limit reached
    ToolChange : BOOL ;	//Tool being changed
    FixedLoc : BOOL ;	//Tool fixed location coded
    ToolUsed : BOOL ;	//Tool was in use
    T_no : INT ;	//Tool new: T no.
    ToolHolder : INT ;	// TH-No as tool compensation reference
    MtMyMag : INT ;	// MtoolNumber the tool is loaded onto
    MtMyPlace : INT ;	// MtoolPlaceNum ~
    IF : ARRAY  [1 .. 7 ] OF STRUCT
     reserved : INT ;	// reserved
    END_STRUCT ;
   END_STRUCT ;
  END_STRUCT ;	
END_TYPE

TYPE UDT 1073
VERSION : 0.0
  STRUCT
   MTIF : ARRAY  [1 .. 16 ] OF STRUCT
    MtType : INT ;
    MtPlaces : INT ;
    MtDistance : REAL ;
    MtNumNew : INT ;	// MT-No. new Tool
    MtPlaceNumNew : INT ;	// MtoolPlaceNum  ~
    MtNumOld : INT ;	// MT-No. old Tool
    MtPlaceNumOld : INT ;	// MtoolPlaceNum  ~
    LocType : INT ;	//Tool new: location type
    SLeft : INT ;	//Tool new: size left
    SRight : INT ;	//Tool new: size right
    STop : INT ;	//Tool new: size top
    SBottom : INT ;	//Tool new: size bottom
    ToolInBuff : BOOL ;	//ID for tools in buffer
    IgnoreDisab : BOOL ;	//Ignore disabled
    TBUnloaded : BOOL ;	//To be unloaded
    TBLoaded : BOOL ;	//To be loaded
    MasterTool : BOOL ;	//Master tool
    n26_5 : BOOL ;	//reserved
    n26_6 : BOOL ;	//reserved
    HandTool : BOOL ;	//Hand tool
    ActTool : BOOL ;	//Active tool
    ToolEnabl : BOOL ;	//Tool enabled
    ToolDisab : BOOL ;	//Tool disabled
    Measured : BOOL ;	//Tool measured
    Prewarn : BOOL ;	//Prewarning limit reached
    ToolChange : BOOL ;	//Tool being changed
    FixedLoc : BOOL ;	//Tool fixed location coded
    ToolUsed : BOOL ;	//Tool was in use
    T_no : INT ;	//Tool new: T no.
    ToolHolder : INT ;	// TH-No as tool compensation reference
    MtMyMag : INT ;	// MtoolNumber the tool is loaded onto
    MtMyPlace : INT ;	// MtoolPlaceNum ~
    IF : ARRAY  [1 .. 7 ] OF STRUCT
     reserved : INT ;	// reserved
    END_STRUCT ;
   END_STRUCT ;
  END_STRUCT ;	
END_TYPE

// FB 1: know-how protected block, not included

// FB 2: know-how protected block, not included

// FB 3: know-how protected block, not included

// FB 4: know-how protected block, not included

// FB 5: know-how protected block, not included

// FB 6: know-how protected block, not included

// FB 7: know-how protected block, not included

// FB 9: know-how protected block, not included

// FB 10: know-how protected block, not included

// FB 11: know-how protected block, not included

// FB 29: know-how protected block, not included

FUNCTION_BLOCK "Table_Ctrl"	// FB 100
AUTHOR : SEDIN
VERSION : 0.1
VAR
  Auxiliary : ARRAY  [0 .. 15 ] OF //Вспомогательная ячейка
  BOOL ;
END_VAR
VAR_TEMP
  ActMoment : INT ;	//Текущий момент, ось 1
END_VAR
BEGIN
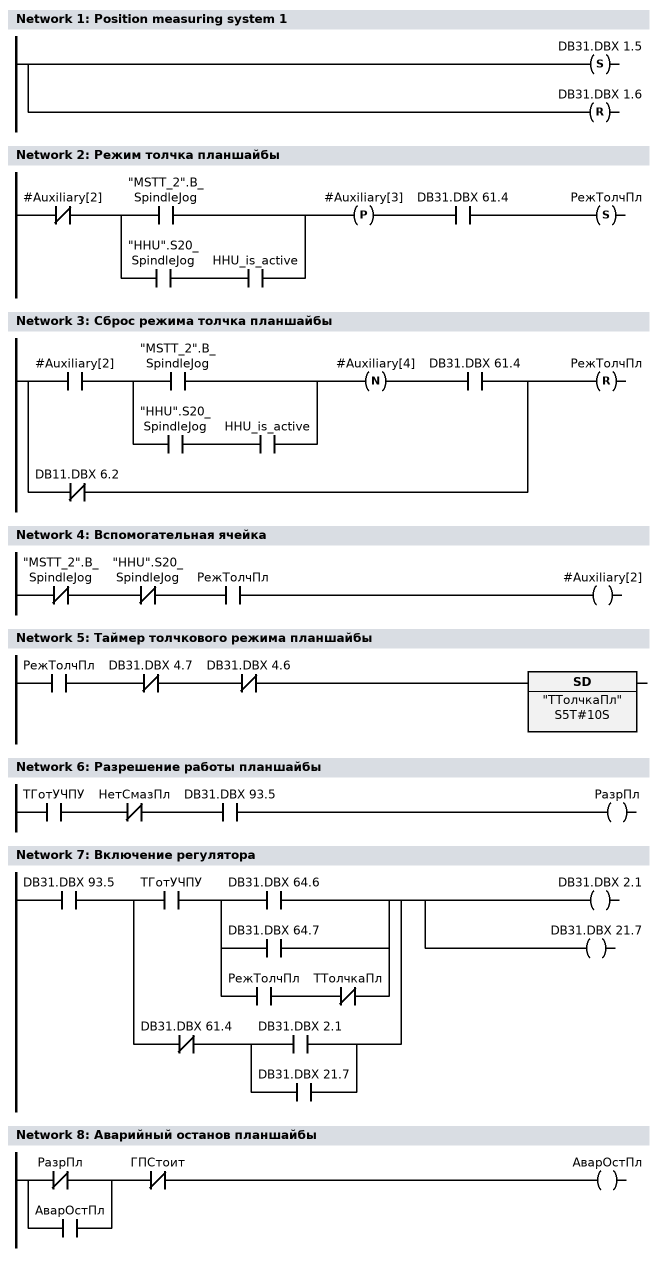
NETWORK
TITLE = Position measuring system 1
      SET;
      S     DB31.DBX 1.5;
      R     DB31.DBX 1.6;
NETWORK
TITLE = Режим толчка планшайбы
      AN    #Auxiliary[2];
      A(;
      O     "MSTT_2".B_SpindleJog;
      O;
      A     "HHU".S20_SpindleJog;
      A     "HHU_is_active";
      );
      FP    #Auxiliary[3];
      A     DB31.DBX 61.4;
      S     "РежТолчПл";
NETWORK
TITLE = Сброс режима толчка планшайбы
      A     #Auxiliary[2];
      A(;
      O     "MSTT_2".B_SpindleJog;
      O;
      A     "HHU".S20_SpindleJog;
      A     "HHU_is_active";
      );
      FN    #Auxiliary[4];
      A     DB31.DBX 61.4;
      ON    DB11.DBX 6.2;
      R     "РежТолчПл";
NETWORK
TITLE = Вспомогательная ячейка
      AN    "MSTT_2".B_SpindleJog;
      AN    "HHU".S20_SpindleJog;
      A     "РежТолчПл";
      =     #Auxiliary[2];
NETWORK
TITLE = Таймер толчкового режима планшайбы
      A     "РежТолчПл";
      AN    DB31.DBX 4.7;
      AN    DB31.DBX 4.6;
      L     S5T#10S;
      SD    "ТТолчкаПл";
NETWORK
TITLE = Разрешение работы планшайбы
      A     "ТГотУЧПУ";
      AN    "НетСмазПл";
      A     DB31.DBX 93.5;
      =     "РазрПл";
NETWORK
TITLE = Включение регулятора
      A     DB31.DBX 93.5;
      A(;
      A     "ТГотУЧПУ";
      A(;
      O     DB31.DBX 64.6;
      O     DB31.DBX 64.7;
      O;
      A     "РежТолчПл";
      AN    "ТТолчкаПл";
      );
      O;
      AN    DB31.DBX 61.4;
      A(;
      O     DB31.DBX 2.1;
      O     DB31.DBX 21.7;
      );
      );
      =     DB31.DBX 2.1;
      =     DB31.DBX 21.7;
NETWORK
TITLE = Аварийный останов планшайбы
      A(;
      ON    "РазрПл";
      O     "АварОстПл";
      );
      AN    "ГПСтоит";
      =     "АварОстПл";
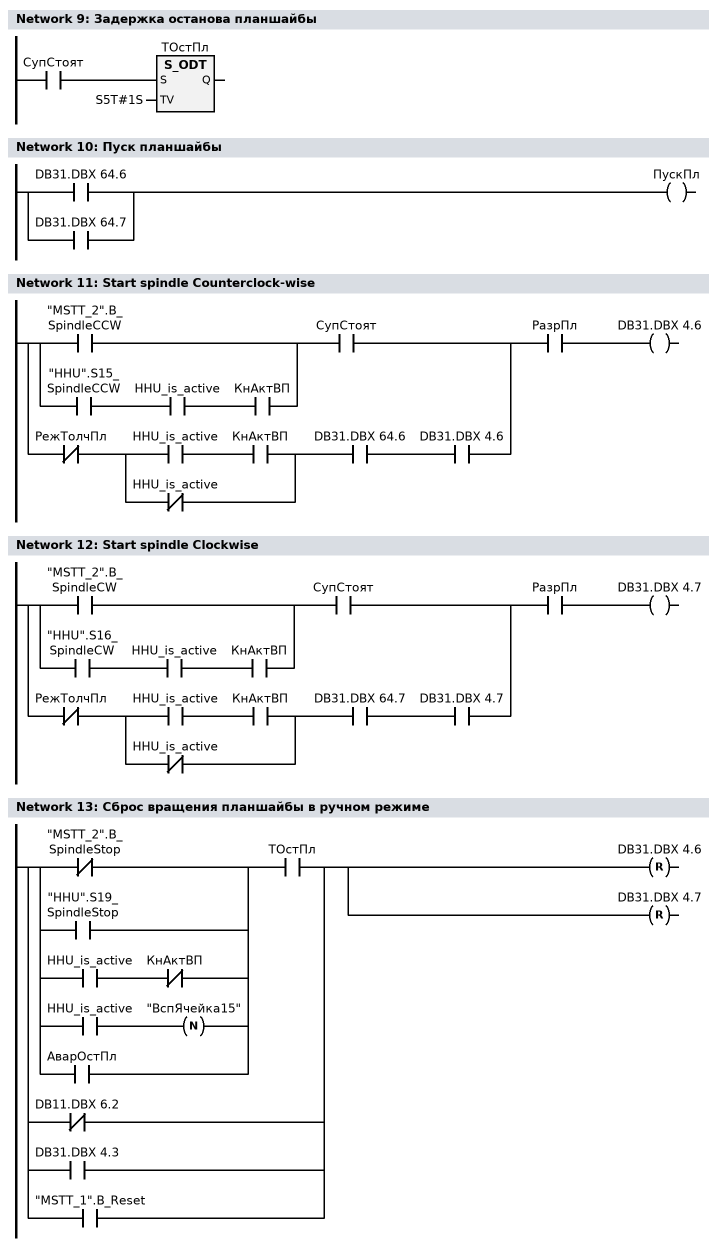
NETWORK
TITLE = Задержка останова планшайбы
      A     "СупСтоят";
      L     S5T#1S;
      SD    "ТОстПл";
      NOP   0;
      NOP   0;
      NOP   0;
      NOP   0;
NETWORK
TITLE = Пуск планшайбы
      O     DB31.DBX 64.6;
      O     DB31.DBX 64.7;
      =     "ПускПл";
NETWORK
TITLE = Start spindle Counterclock-wise
      A(;
      A(;
      O     "MSTT_2".B_SpindleCCW;
      O;
      A     "HHU".S15_SpindleCCW;
      A     "HHU_is_active";
      A     "КнАктВП";
      );
      A     "СупСтоят";
      O;
      AN    "РежТолчПл";
      A(;
      A     "HHU_is_active";
      A     "КнАктВП";
      ON    "HHU_is_active";
      );
      A     DB31.DBX 64.6;
      A     DB31.DBX 4.6;
      );
      A     "РазрПл";
      =     DB31.DBX 4.6;
NETWORK
TITLE = Start spindle Clockwise
      A(;
      A(;
      O     "MSTT_2".B_SpindleCW;
      O;
      A     "HHU".S16_SpindleCW;
      A     "HHU_is_active";
      A     "КнАктВП";
      );
      A     "СупСтоят";
      O;
      AN    "РежТолчПл";
      A(;
      A     "HHU_is_active";
      A     "КнАктВП";
      ON    "HHU_is_active";
      );
      A     DB31.DBX 64.7;
      A     DB31.DBX 4.7;
      );
      A     "РазрПл";
      =     DB31.DBX 4.7;
NETWORK
TITLE = Сброс вращения планшайбы в ручном режиме
      A(;
      ON    "MSTT_2".B_SpindleStop;
      O     "HHU".S19_SpindleStop;
      O(;
      A     "HHU_is_active";
      AN    "КнАктВП";
      );
      O(;
      A     "HHU_is_active";
      FN    "ВспЯчейка15";
      );
      O     "АварОстПл";
      );
      A     "ТОстПл";
      ON    DB11.DBX 6.2;
      O     DB31.DBX 4.3;
      O     "MSTT_1".B_Reset;
      R     DB31.DBX 4.6;
      R     DB31.DBX 4.7;
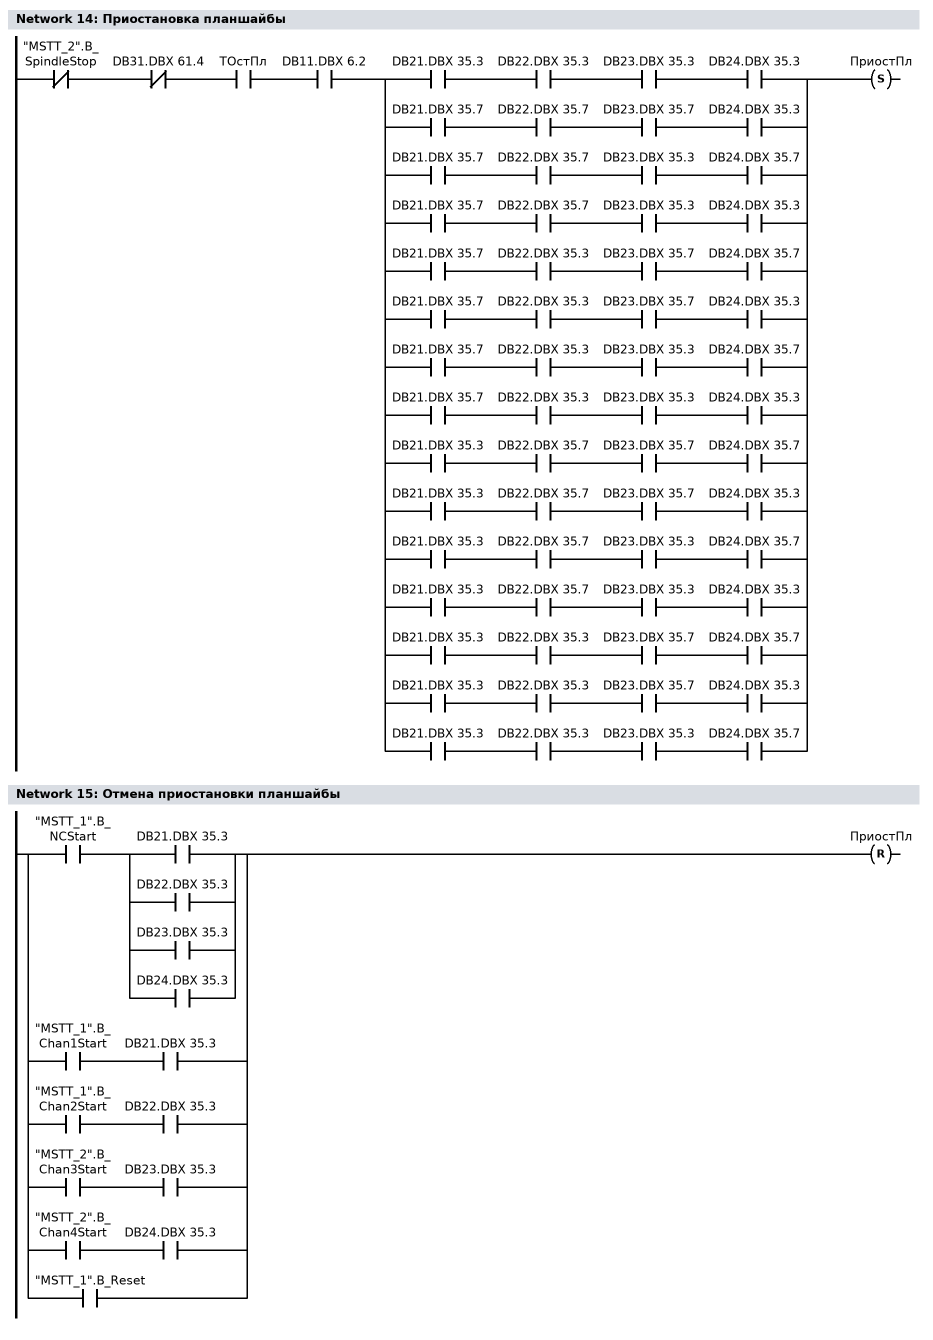
NETWORK
TITLE = Приостановка планшайбы
      AN    "MSTT_2".B_SpindleStop;
      AN    DB31.DBX 61.4;
      A     "ТОстПл";
      A     DB11.DBX 6.2;
      A(;
      A     DB21.DBX 35.3;
      A     DB22.DBX 35.3;
      A     DB23.DBX 35.3;
      A     DB24.DBX 35.3;
      O;
      A     DB21.DBX 35.7;
      A     DB22.DBX 35.7;
      A     DB23.DBX 35.7;
      A     DB24.DBX 35.3;
      O;
      A     DB21.DBX 35.7;
      A     DB22.DBX 35.7;
      A     DB23.DBX 35.3;
      A     DB24.DBX 35.7;
      O;
      A     DB21.DBX 35.7;
      A     DB22.DBX 35.7;
      A     DB23.DBX 35.3;
      A     DB24.DBX 35.3;
      O;
      A     DB21.DBX 35.7;
      A     DB22.DBX 35.3;
      A     DB23.DBX 35.7;
      A     DB24.DBX 35.7;
      O;
      A     DB21.DBX 35.7;
      A     DB22.DBX 35.3;
      A     DB23.DBX 35.7;
      A     DB24.DBX 35.3;
      O;
      A     DB21.DBX 35.7;
      A     DB22.DBX 35.3;
      A     DB23.DBX 35.3;
      A     DB24.DBX 35.7;
      O;
      A     DB21.DBX 35.7;
      A     DB22.DBX 35.3;
      A     DB23.DBX 35.3;
      A     DB24.DBX 35.3;
      O;
      A     DB21.DBX 35.3;
      A     DB22.DBX 35.7;
      A     DB23.DBX 35.7;
      A     DB24.DBX 35.7;
      O;
      A     DB21.DBX 35.3;
      A     DB22.DBX 35.7;
      A     DB23.DBX 35.7;
      A     DB24.DBX 35.3;
      O;
      A     DB21.DBX 35.3;
      A     DB22.DBX 35.7;
      A     DB23.DBX 35.3;
      A     DB24.DBX 35.7;
      O;
      A     DB21.DBX 35.3;
      A     DB22.DBX 35.7;
      A     DB23.DBX 35.3;
      A     DB24.DBX 35.3;
      O;
      A     DB21.DBX 35.3;
      A     DB22.DBX 35.3;
      A     DB23.DBX 35.7;
      A     DB24.DBX 35.7;
      O;
      A     DB21.DBX 35.3;
      A     DB22.DBX 35.3;
      A     DB23.DBX 35.7;
      A     DB24.DBX 35.3;
      O;
      A     DB21.DBX 35.3;
      A     DB22.DBX 35.3;
      A     DB23.DBX 35.3;
      A     DB24.DBX 35.7;
      );
      S     "ПриостПл";
NETWORK
TITLE = Отмена приостановки планшайбы
      A     "MSTT_1".B_NCStart;
      A(;
      O     DB21.DBX 35.3;
      O     DB22.DBX 35.3;
      O     DB23.DBX 35.3;
      O     DB24.DBX 35.3;
      );
      O;
      A     "MSTT_1".B_Chan1Start;
      A     DB21.DBX 35.3;
      O;
      A     "MSTT_1".B_Chan2Start;
      A     DB22.DBX 35.3;
      O;
      A     "MSTT_2".B_Chan3Start;
      A     DB23.DBX 35.3;
      O;
      A     "MSTT_2".B_Chan4Start;
      A     DB24.DBX 35.3;
      O     "MSTT_1".B_Reset;
      R     "ПриостПл";
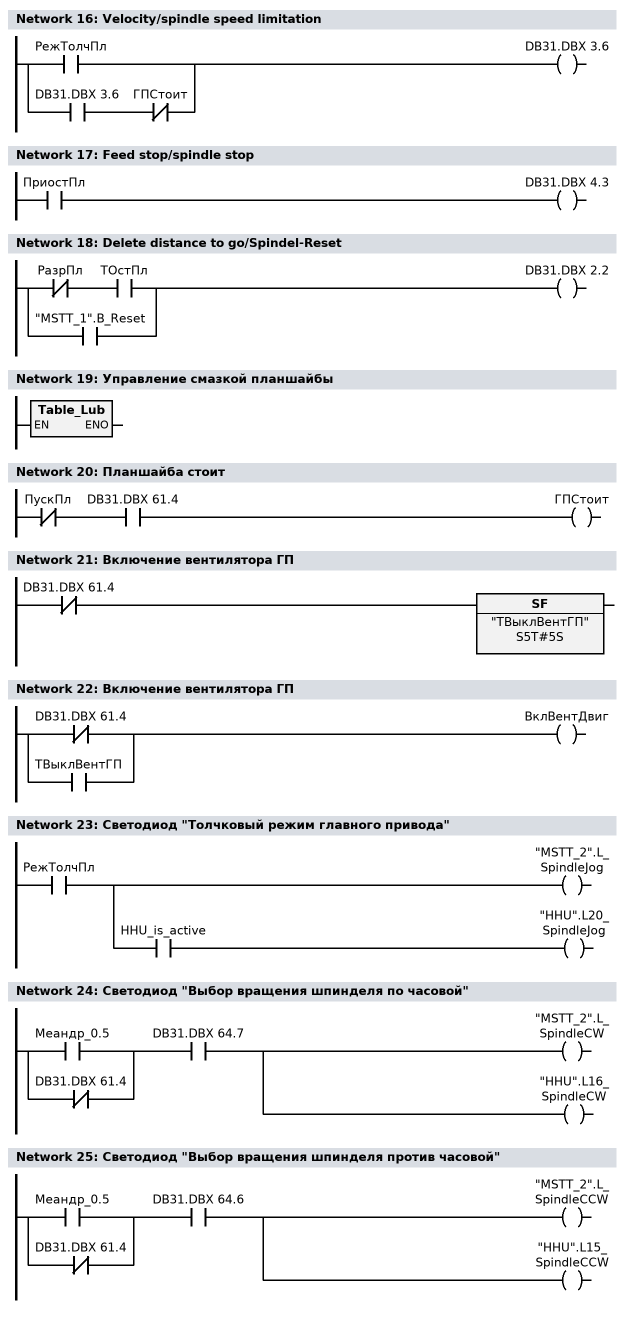
NETWORK
TITLE = Velocity/spindle speed limitation
      O     "РежТолчПл";
      O;
      A     DB31.DBX 3.6;
      AN    "ГПСтоит";
      =     DB31.DBX 3.6;
NETWORK
TITLE = Feed stop/spindle stop
      A     "ПриостПл";
      =     DB31.DBX 4.3;
NETWORK
TITLE = Delete distance to go/Spindel-Reset
      AN    "РазрПл";
      A     "ТОстПл";
      O     "MSTT_1".B_Reset;
      =     DB31.DBX 2.2;
NETWORK
TITLE = Управление смазкой планшайбы
      CALL  "Table_Lub";
      NOP   0;
NETWORK
TITLE = Планшайба стоит
      AN    "ПускПл";
      A     DB31.DBX 61.4;
      =     "ГПСтоит";
NETWORK
TITLE = Включение вентилятора ГП
      AN    DB31.DBX 61.4;
      L     S5T#5S;
      SF    "ТВыклВентГП";
NETWORK
TITLE = Включение вентилятора ГП
      ON    DB31.DBX 61.4;
      O     "ТВыклВентГП";
      =     "ВклВентДвиг";
NETWORK
TITLE = Светодиод "Толчковый режим главного привода"
      A     "РежТолчПл";
      =     L 2.0;
      A     L 2.0;
      BLD   102;
      =     "MSTT_2".L_SpindleJog;
      A     L 2.0;
      A     "HHU_is_active";
      =     "HHU".L20_SpindleJog;
NETWORK
TITLE = Светодиод "Выбор вращения шпинделя по часовой"
      A(;
      O     "Меандр_0.5";
      ON    DB31.DBX 61.4;
      );
      A     DB31.DBX 64.7;
      =     "MSTT_2".L_SpindleCW;
      =     "HHU".L16_SpindleCW;
NETWORK
TITLE = Светодиод "Выбор вращения шпинделя против часовой"
      A(;
      O     "Меандр_0.5";
      ON    DB31.DBX 61.4;
      );
      A     DB31.DBX 64.6;
      =     "MSTT_2".L_SpindleCCW;
      =     "HHU".L15_SpindleCCW;
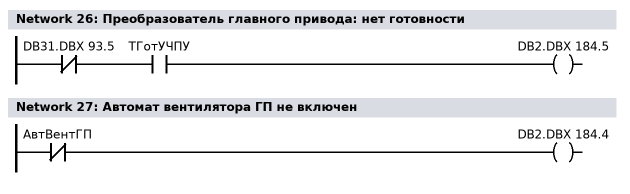
NETWORK
TITLE = Преобразователь главного привода: нет готовности
      AN    DB31.DBX 93.5;
      A     "ТГотУЧПУ";
      =     DB2.DBX 184.5;
NETWORK
TITLE = Автомат вентилятора ГП не включен
      AN    "АвтВентГП";
      =     DB2.DBX 184.4;
END_FUNCTION_BLOCK

FUNCTION_BLOCK "Support1_Ctrl"	// FB 101
AUTHOR : SEDIN
VERSION : 0.1
VAR
  Auxiliary : ARRAY  [0 .. 15 ] OF //Вспомогательная ячейка
  BOOL ;
  Unbrake1 : BOOL ;	//Требование разжима оси 1
  Unbrake2 : BOOL ;	//Требование разжима оси 2
  ErrorLub : BOOL ;	//Ошибка ИСС
  Sup_Lub : FB 121;	//Управление смазкой суппорта
  StartFC18_1 : BOOL ;	//Старт FC18
  StopFC18_1 : BOOL ;	//Остановка FC18
  InPosFC18_1 : BOOL ;	//Выполнение FC18
  ErrorFC18_1 : BOOL ;	//Ошибка FC18
  StartFC18_2 : BOOL ;	//Старт FC18
  StopFC18_2 : BOOL ;	//Остановка FC18
  InPosFC18_2 : BOOL ;	//Выполнение FC18
  ErrorFC18_2 : BOOL ;	//Ошибка FC18
  StateFC18_1 : BYTE ;	//Состояние FC18
  StateFC18_2 : BYTE ;	//Состояние FC18
END_VAR
VAR_TEMP
  Permission : BOOL ;	//Разрешение работы суппорта
  Permission1 : BOOL ;	//Разрешение работы суппорта, ось 1
  Permission2 : BOOL ;	//Разрешение работы суппорта, ось 2
  JogStop : BOOL ;	//Останов подачи в ручном режиме
  Stop1 : BOOL ;	//Суппорт стоит, ось 1
  Stop2 : BOOL ;	//Суппорт стоит, ось 2
  ErrorLub1 : BOOL ;	//Низкий уровень масла в ИСС
  ErrorLub2 : BOOL ;	//Не достигнуто давление в ИСС
  ErrorLub3 : BOOL ;	//Нет падения давления в ИСС
END_VAR
BEGIN
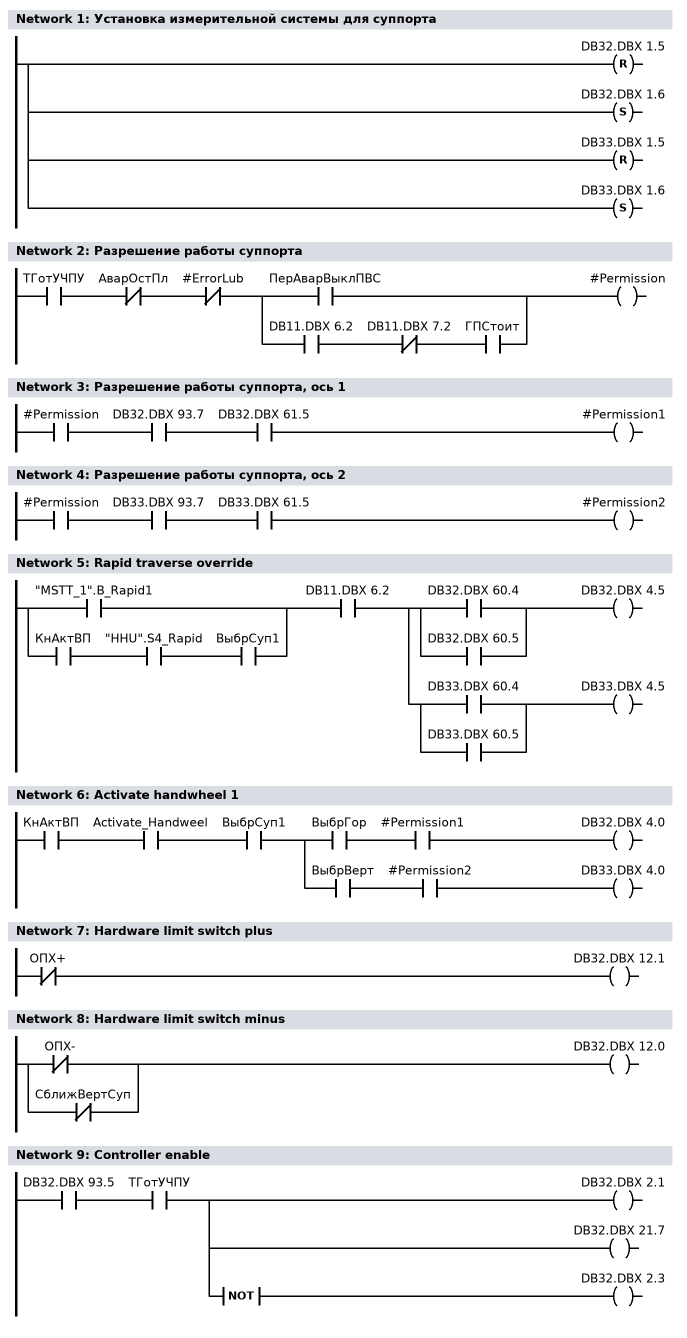
NETWORK
TITLE = Установка измерительной системы для суппорта
      SET;
      R     DB32.DBX 1.5;
      S     DB32.DBX 1.6;
      R     DB33.DBX 1.5;
      S     DB33.DBX 1.6;
NETWORK
TITLE = Разрешение работы суппорта
      A     "ТГотУЧПУ";
      AN    "АварОстПл";
      AN    #ErrorLub;
      A(;
      O     "ПерАварВыклПВС";
      O;
      A     DB11.DBX 6.2;
      AN    DB11.DBX 7.2;
      A     "ГПСтоит";
      );
      =     #Permission;
NETWORK
TITLE = Разрешение работы суппорта, ось 1
      A     #Permission;
      A     DB32.DBX 93.7;
      A     DB32.DBX 61.5;
      =     #Permission1;
NETWORK
TITLE = Разрешение работы суппорта, ось 2
      A     #Permission;
      A     DB33.DBX 93.7;
      A     DB33.DBX 61.5;
      =     #Permission2;
NETWORK
TITLE = Rapid traverse override
      A(;
      O     "MSTT_1".B_Rapid1;
      O;
      A     "КнАктВП";
      A     "HHU".S4_Rapid;
      A     "ВыбрСуп1";
      );
      A     DB11.DBX 6.2;
      =     L 2.0;
      A     L 2.0;
      A(;
      O     DB32.DBX 60.4;
      O     DB32.DBX 60.5;
      );
      =     DB32.DBX 4.5;
      A     L 2.0;
      A(;
      O     DB33.DBX 60.4;
      O     DB33.DBX 60.5;
      );
      =     DB33.DBX 4.5;
NETWORK
TITLE = Activate handwheel 1
      A     "КнАктВП";
      A     "Activate_Handweel";
      A     "ВыбрСуп1";
      =     L 2.0;
      A     L 2.0;
      A     "ВыбрГор";
      A     #Permission1;
      =     DB32.DBX 4.0;
      A     L 2.0;
      A     "ВыбрВерт";
      A     #Permission2;
      =     DB33.DBX 4.0;
NETWORK
TITLE = Hardware limit switch plus
      AN    "ОПX+";
      =     DB32.DBX 12.1;
NETWORK
TITLE = Hardware limit switch minus
      ON    "ОПX-";
      ON    "СближВертСуп";
      =     DB32.DBX 12.0;
NETWORK
TITLE = Controller enable
      A     DB32.DBX 93.5;
      A     "ТГотУЧПУ";
      =     L 2.0;
      A     L 2.0;
      BLD   102;
      =     DB32.DBX 2.1;
      A     L 2.0;
      BLD   102;
      =     DB32.DBX 21.7;
      A     L 2.0;
      NOT;
      =     DB32.DBX 2.3;
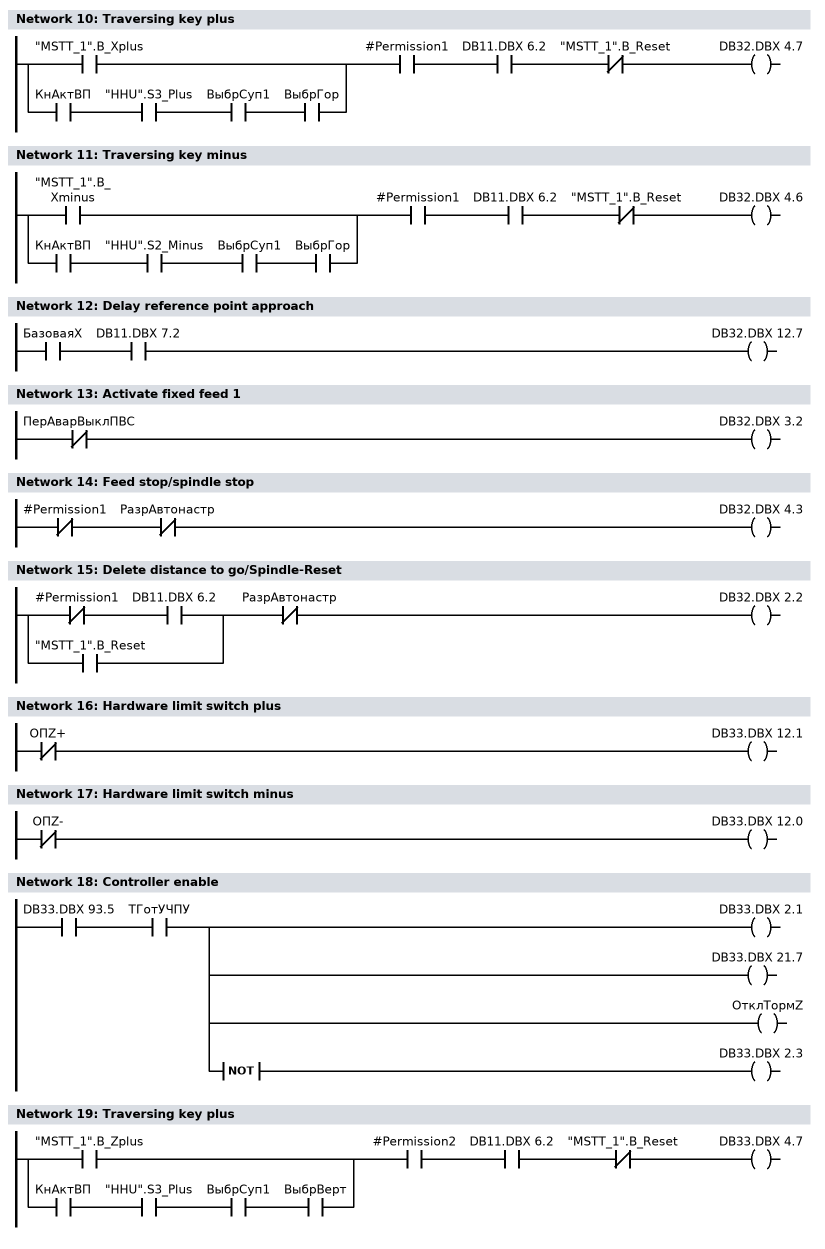
NETWORK
TITLE = Traversing key plus
      A(;
      O     "MSTT_1".B_Xplus;
      O;
      A     "КнАктВП";
      A     "HHU".S3_Plus;
      A     "ВыбрСуп1";
      A     "ВыбрГор";
      );
      A     #Permission1;
      A     DB11.DBX 6.2;
      AN    "MSTT_1".B_Reset;
      =     DB32.DBX 4.7;
NETWORK
TITLE = Traversing key minus
      A(;
      O     "MSTT_1".B_Xminus;
      O;
      A     "КнАктВП";
      A     "HHU".S2_Minus;
      A     "ВыбрСуп1";
      A     "ВыбрГор";
      );
      A     #Permission1;
      A     DB11.DBX 6.2;
      AN    "MSTT_1".B_Reset;
      =     DB32.DBX 4.6;
NETWORK
TITLE = Delay reference point approach
      A     "БазоваяX";
      A     DB11.DBX 7.2;
      =     DB32.DBX 12.7;
NETWORK
TITLE = Activate fixed feed 1
      AN    "ПерАварВыклПВС";
      =     DB32.DBX 3.2;
NETWORK
TITLE = Feed stop/spindle stop
      AN    #Permission1;
      AN    "РазрАвтонастр";
      =     DB32.DBX 4.3;
NETWORK
TITLE = Delete distance to go/Spindle-Reset
      A(;
      AN    #Permission1;
      A     DB11.DBX 6.2;
      O     "MSTT_1".B_Reset;
      );
      AN    "РазрАвтонастр";
      =     DB32.DBX 2.2;
NETWORK
TITLE = Hardware limit switch plus
      AN    "ОПZ+";
      =     DB33.DBX 12.1;
NETWORK
TITLE = Hardware limit switch minus
      AN    "ОПZ-";
      =     DB33.DBX 12.0;
NETWORK
TITLE = Controller enable
      A     DB33.DBX 93.5;
      A     "ТГотУЧПУ";
      =     L 2.0;
      A     L 2.0;
      BLD   102;
      =     DB33.DBX 2.1;
      A     L 2.0;
      BLD   102;
      =     DB33.DBX 21.7;
      A     L 2.0;
      BLD   102;
      =     "ОтклТормZ";
      A     L 2.0;
      NOT;
      =     DB33.DBX 2.3;
NETWORK
TITLE = Traversing key plus
      A(;
      O     "MSTT_1".B_Zplus;
      O;
      A     "КнАктВП";
      A     "HHU".S3_Plus;
      A     "ВыбрСуп1";
      A     "ВыбрВерт";
      );
      A     #Permission2;
      A     DB11.DBX 6.2;
      AN    "MSTT_1".B_Reset;
      =     DB33.DBX 4.7;
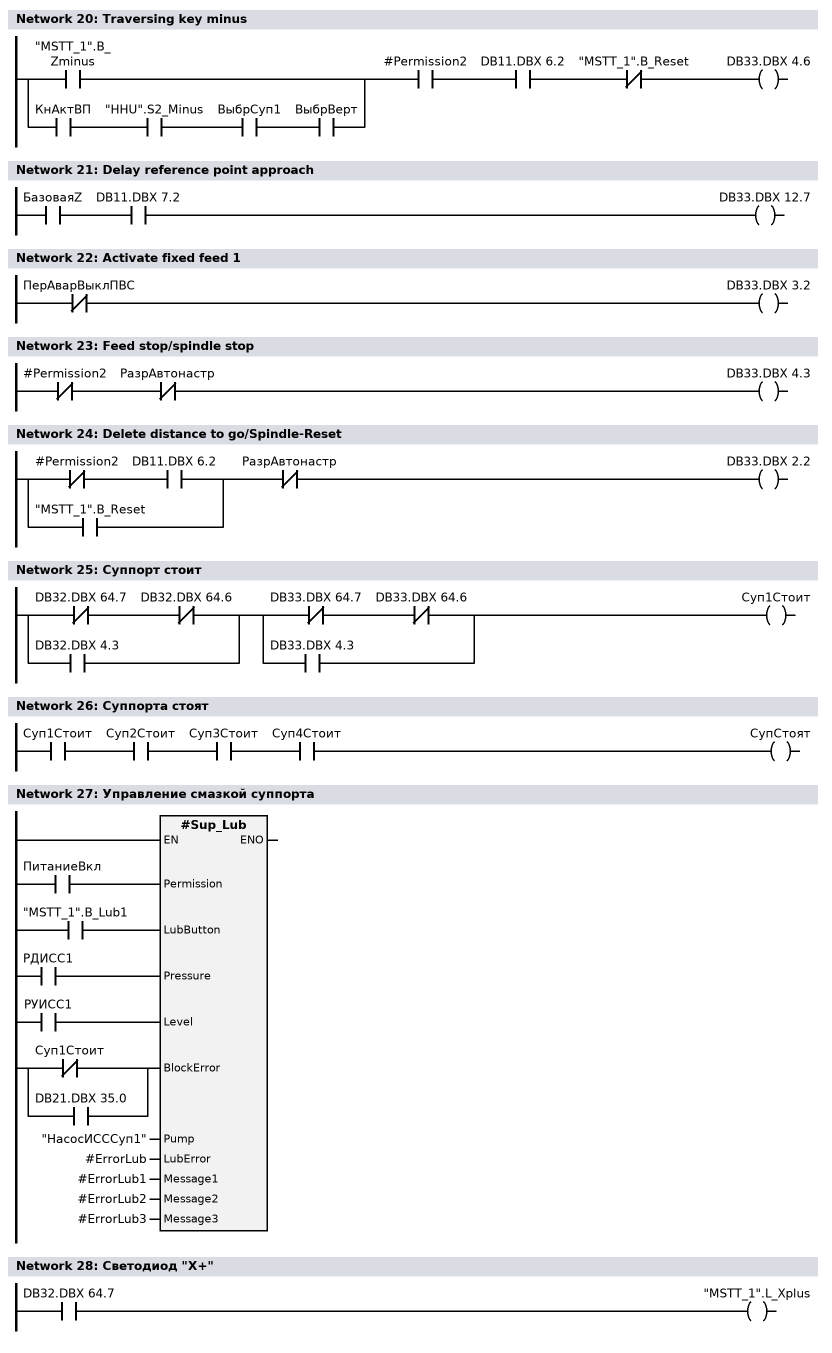
NETWORK
TITLE = Traversing key minus
      A(;
      O     "MSTT_1".B_Zminus;
      O;
      A     "КнАктВП";
      A     "HHU".S2_Minus;
      A     "ВыбрСуп1";
      A     "ВыбрВерт";
      );
      A     #Permission2;
      A     DB11.DBX 6.2;
      AN    "MSTT_1".B_Reset;
      =     DB33.DBX 4.6;
NETWORK
TITLE = Delay reference point approach
      A     "БазоваяZ";
      A     DB11.DBX 7.2;
      =     DB33.DBX 12.7;
NETWORK
TITLE = Activate fixed feed 1
      AN    "ПерАварВыклПВС";
      =     DB33.DBX 3.2;
NETWORK
TITLE = Feed stop/spindle stop
      AN    #Permission2;
      AN    "РазрАвтонастр";
      =     DB33.DBX 4.3;
NETWORK
TITLE = Delete distance to go/Spindle-Reset
      A(;
      AN    #Permission2;
      A     DB11.DBX 6.2;
      O     "MSTT_1".B_Reset;
      );
      AN    "РазрАвтонастр";
      =     DB33.DBX 2.2;
NETWORK
TITLE = Суппорт стоит
      A(;
      AN    DB32.DBX 64.7;
      AN    DB32.DBX 64.6;
      O     DB32.DBX 4.3;
      );
      A(;
      AN    DB33.DBX 64.7;
      AN    DB33.DBX 64.6;
      O     DB33.DBX 4.3;
      );
      =     "Суп1Стоит";
NETWORK
TITLE = Суппорта стоят
      A     "Суп1Стоит";
      A     "Суп2Стоит";
      A     "Суп3Стоит";
      A     "Суп4Стоит";
      =     "СупСтоят";
NETWORK
TITLE = Управление смазкой суппорта
      A     "ПитаниеВкл";
      =     L 2.0;
      BLD   103;
      A     "MSTT_1".B_Lub1;
      =     L 2.1;
      BLD   103;
      A     "РДИСС1";
      =     L 2.2;
      BLD   103;
      A     "РУИСС1";
      =     L 2.3;
      BLD   103;
      A(;
      ON    "Суп1Стоит";
      O     DB21.DBX 35.0;
      );
      =     L 2.4;
      BLD   103;
      CALL  #Sup_Lub (
           Permission               := L 2.0,
           LubButton                := L 2.1,
           Pressure                 := L 2.2,
           Level                    := L 2.3,
           BlockError               := L 2.4,
           Pump                     := "НасосИСССуп1",
           LubError                 := #ErrorLub,
           Message1                 := #ErrorLub1,
           Message2                 := #ErrorLub2,
           Message3                 := #ErrorLub3);
      NOP   0;
NETWORK
TITLE = Светодиод "X+"
      A     DB32.DBX 64.7;
      =     "MSTT_1".L_Xplus;
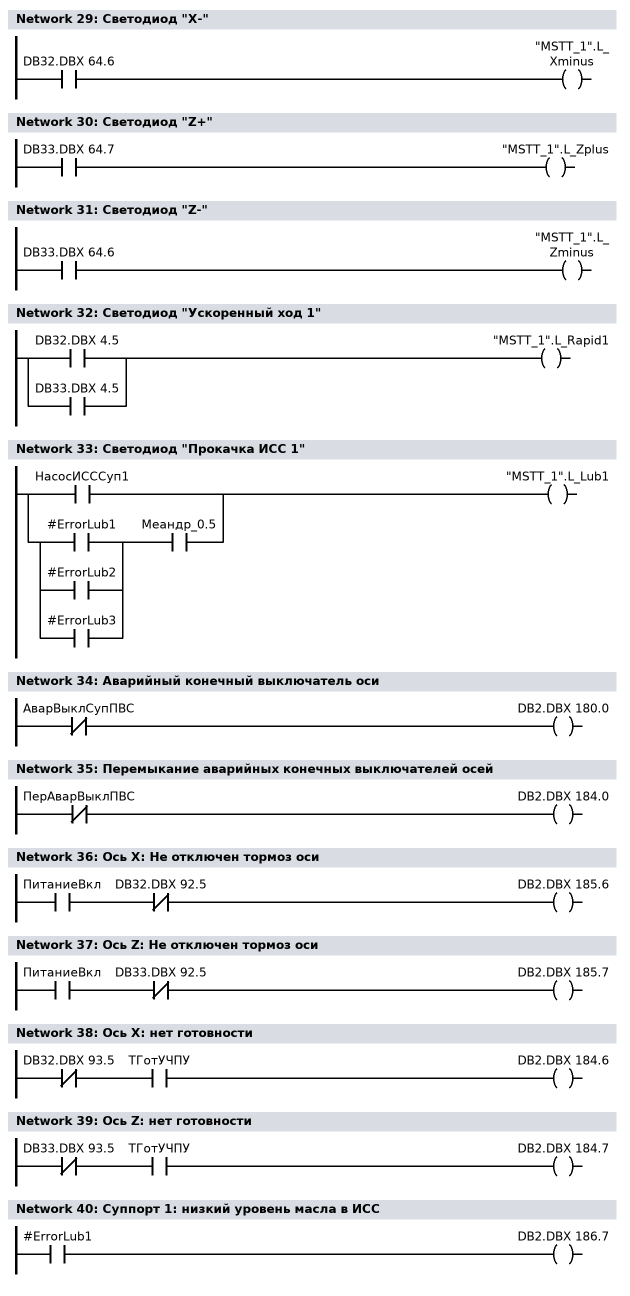
NETWORK
TITLE = Светодиод "X-"
      A     DB32.DBX 64.6;
      =     "MSTT_1".L_Xminus;
NETWORK
TITLE = Светодиод "Z+"
      A     DB33.DBX 64.7;
      =     "MSTT_1".L_Zplus;
NETWORK
TITLE = Светодиод "Z-"
      A     DB33.DBX 64.6;
      =     "MSTT_1".L_Zminus;
NETWORK
TITLE = Светодиод "Ускоренный ход 1"
      O     DB32.DBX 4.5;
      O     DB33.DBX 4.5;
      =     "MSTT_1".L_Rapid1;
NETWORK
TITLE = Светодиод "Прокачка ИСС 1"
      O     "НасосИСССуп1";
      O;
      A(;
      O     #ErrorLub1;
      O     #ErrorLub2;
      O     #ErrorLub3;
      );
      A     "Меандр_0.5";
      =     "MSTT_1".L_Lub1;
NETWORK
TITLE = Аварийный конечный выключатель оси
      AN    "АварВыклСупПВС";
      =     DB2.DBX 180.0;
NETWORK
TITLE = Перемыкание аварийных конечных выключателей осей
      AN    "ПерАварВыклПВС";
      =     DB2.DBX 184.0;
NETWORK
TITLE = Ось X: Не отключен тормоз оси
      A     "ПитаниеВкл";
      AN    DB32.DBX 92.5;
      =     DB2.DBX 185.6;
NETWORK
TITLE = Ось Z: Не отключен тормоз оси
      A     "ПитаниеВкл";
      AN    DB33.DBX 92.5;
      =     DB2.DBX 185.7;
NETWORK
TITLE = Ось X: нет готовности
      AN    DB32.DBX 93.5;
      A     "ТГотУЧПУ";
      =     DB2.DBX 184.6;
NETWORK
TITLE = Ось Z: нет готовности
      AN    DB33.DBX 93.5;
      A     "ТГотУЧПУ";
      =     DB2.DBX 184.7;
NETWORK
TITLE = Суппорт 1: низкий уровень масла в ИСС 
      A     #ErrorLub1;
      =     DB2.DBX 186.7;
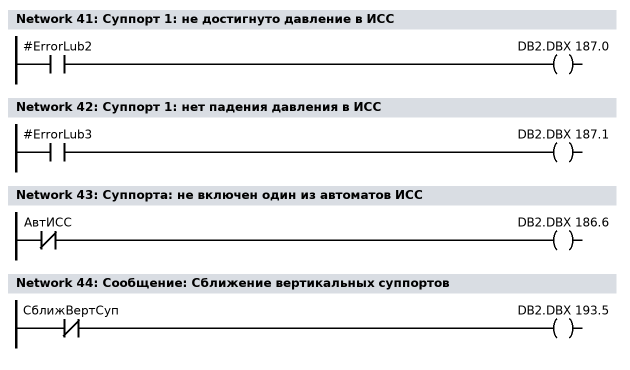
NETWORK
TITLE = Суппорт 1: не достигнуто давление в ИСС
      A     #ErrorLub2;
      =     DB2.DBX 187.0;
NETWORK
TITLE = Суппорт 1: нет падения давления в ИСС
      A     #ErrorLub3;
      =     DB2.DBX 187.1;
NETWORK
TITLE = Суппорта: не включен один из автоматов ИСС
      AN    "АвтИСС";
      =     DB2.DBX 186.6;
NETWORK
TITLE = Сообщение: Сближение вертикальных суппортов
      AN    "СближВертСуп";
      =     DB2.DBX 193.5;
END_FUNCTION_BLOCK

FUNCTION_BLOCK "Support2_Ctrl"	// FB 102
AUTHOR : SEDIN
VERSION : 0.1
VAR
  Auxiliary : ARRAY  [0 .. 15 ] OF //Вспомогательная ячейка
  BOOL ;
  Unbrake1 : BOOL ;	//Требование разжима оси 1
  Unbrake2 : BOOL ;	//Требование разжима оси 2
  ErrorLub : BOOL ;	//Ошибка ИСС
  Sup_Lub : FB 121;	//Управление смазкой суппорта
  StartFC18_1 : BOOL ;	//Старт FC18
  StopFC18_1 : BOOL ;	//Остановка FC18
  InPosFC18_1 : BOOL ;	//Выполнение FC18
  ErrorFC18_1 : BOOL ;	//Ошибка FC18
  StartFC18_2 : BOOL ;	//Старт FC18
  StopFC18_2 : BOOL ;	//Остановка FC18
  InPosFC18_2 : BOOL ;	//Выполнение FC18
  ErrorFC18_2 : BOOL ;	//Ошибка FC18
  StateFC18_1 : BYTE ;	//Состояние FC18
  StateFC18_2 : BYTE ;	//Состояние FC18
END_VAR
VAR_TEMP
  Permission : BOOL ;	//Разрешение работы суппорта
  Permission1 : BOOL ;	//Разрешение работы суппорта, ось 1
  Permission2 : BOOL ;	//Разрешение работы суппорта, ось 2
  JogStop : BOOL ;	//Останов подачи в ручном режиме
  Stop1 : BOOL ;	//Суппорт стоит, ось 1
  Stop2 : BOOL ;	//Суппорт стоит, ось 2
  ErrorLub1 : BOOL ;	//Низкий уровень масла в ИСС
  ErrorLub2 : BOOL ;	//Не достигнуто давление в ИСС
  ErrorLub3 : BOOL ;	//Нет падения давления в ИСС
  GAct : INT ;	//Текущая G-функция 15 группы
END_VAR
BEGIN
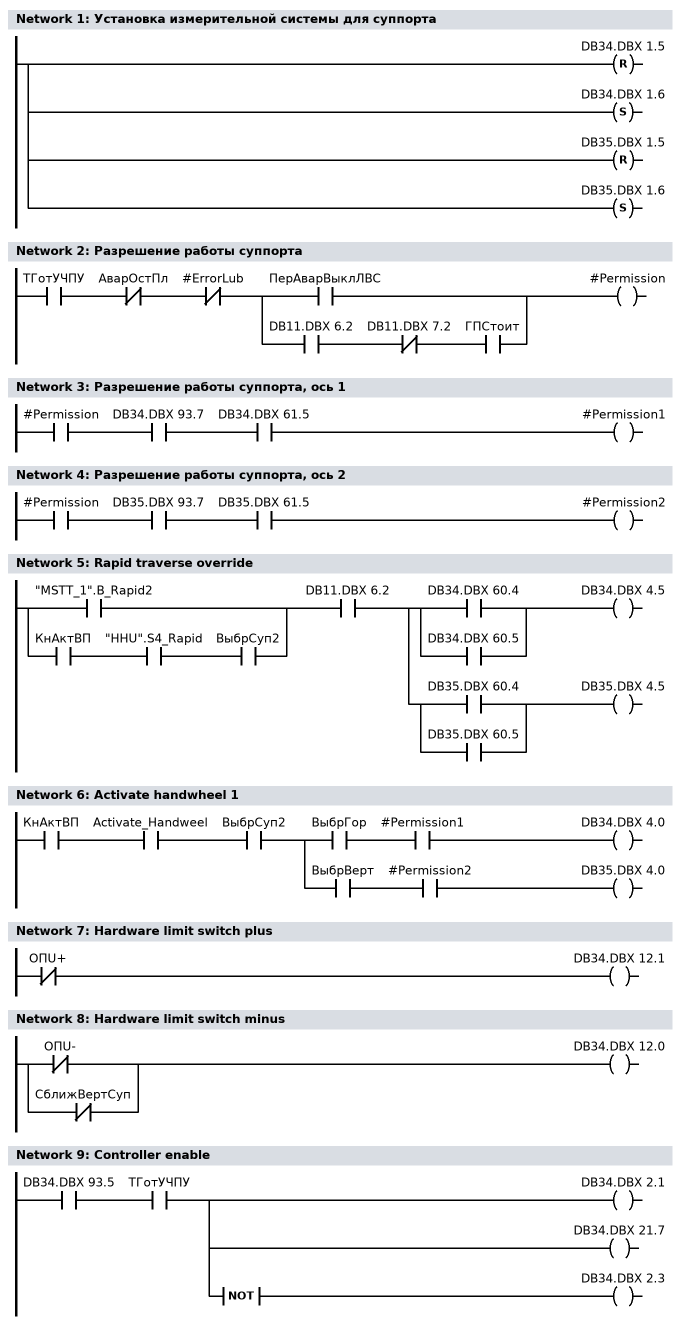
NETWORK
TITLE = Установка измерительной системы для суппорта
      SET;
      R     DB34.DBX 1.5;
      S     DB34.DBX 1.6;
      R     DB35.DBX 1.5;
      S     DB35.DBX 1.6;
NETWORK
TITLE = Разрешение работы суппорта
      A     "ТГотУЧПУ";
      AN    "АварОстПл";
      AN    #ErrorLub;
      A(;
      O     "ПерАварВыклЛВС";
      O;
      A     DB11.DBX 6.2;
      AN    DB11.DBX 7.2;
      A     "ГПСтоит";
      );
      =     #Permission;
NETWORK
TITLE = Разрешение работы суппорта, ось 1
      A     #Permission;
      A     DB34.DBX 93.7;
      A     DB34.DBX 61.5;
      =     #Permission1;
NETWORK
TITLE = Разрешение работы суппорта, ось 2
      A     #Permission;
      A     DB35.DBX 93.7;
      A     DB35.DBX 61.5;
      =     #Permission2;
NETWORK
TITLE = Rapid traverse override
      A(;
      O     "MSTT_1".B_Rapid2;
      O;
      A     "КнАктВП";
      A     "HHU".S4_Rapid;
      A     "ВыбрСуп2";
      );
      A     DB11.DBX 6.2;
      =     L 4.0;
      A     L 4.0;
      A(;
      O     DB34.DBX 60.4;
      O     DB34.DBX 60.5;
      );
      =     DB34.DBX 4.5;
      A     L 4.0;
      A(;
      O     DB35.DBX 60.4;
      O     DB35.DBX 60.5;
      );
      =     DB35.DBX 4.5;
NETWORK
TITLE = Activate handwheel 1
      A     "КнАктВП";
      A     "Activate_Handweel";
      A     "ВыбрСуп2";
      =     L 4.0;
      A     L 4.0;
      A     "ВыбрГор";
      A     #Permission1;
      =     DB34.DBX 4.0;
      A     L 4.0;
      A     "ВыбрВерт";
      A     #Permission2;
      =     DB35.DBX 4.0;
NETWORK
TITLE = Hardware limit switch plus
      AN    "ОПU+";
      =     DB34.DBX 12.1;
NETWORK
TITLE = Hardware limit switch minus
      ON    "ОПU-";
      ON    "СближВертСуп";
      =     DB34.DBX 12.0;
NETWORK
TITLE = Controller enable
      A     DB34.DBX 93.5;
      A     "ТГотУЧПУ";
      =     L 4.0;
      A     L 4.0;
      BLD   102;
      =     DB34.DBX 2.1;
      A     L 4.0;
      BLD   102;
      =     DB34.DBX 21.7;
      A     L 4.0;
      NOT;
      =     DB34.DBX 2.3;
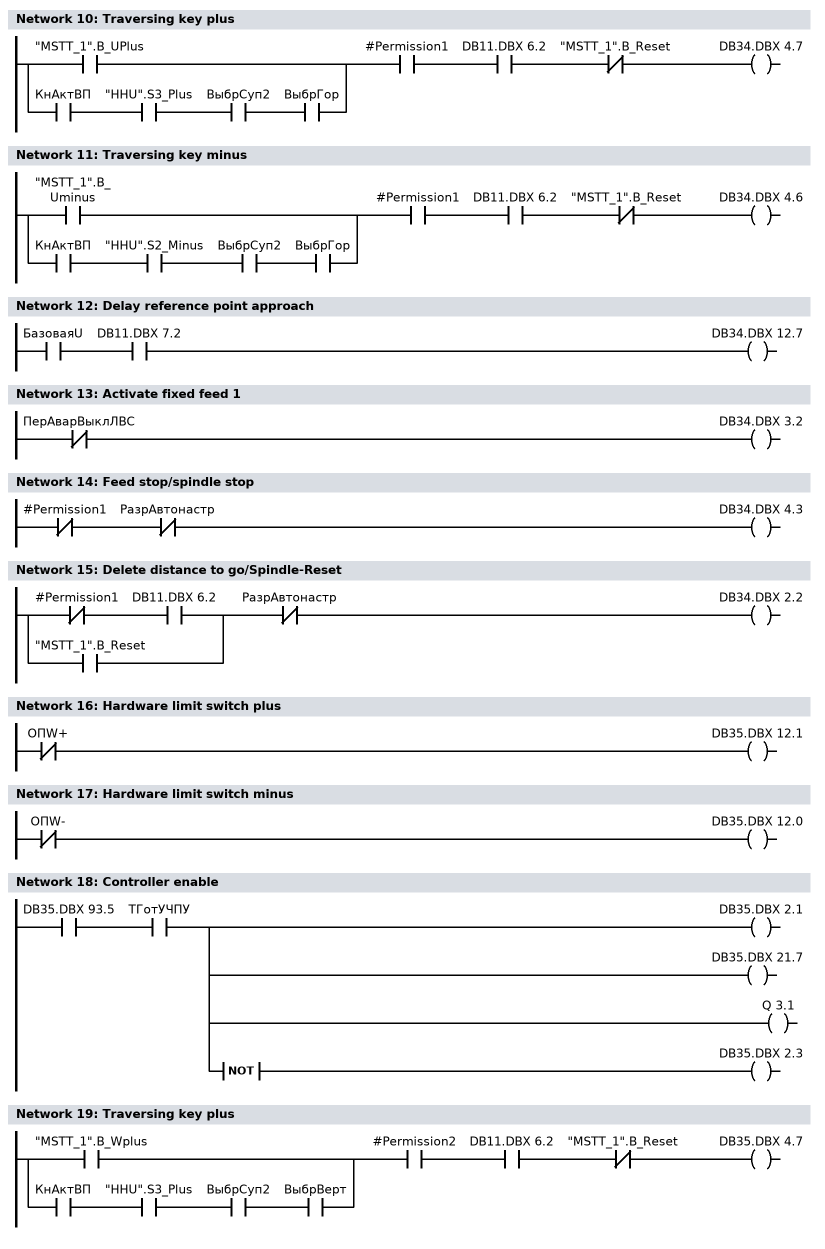
NETWORK
TITLE = Traversing key plus
      A(;
      O     "MSTT_1".B_UPlus;
      O;
      A     "КнАктВП";
      A     "HHU".S3_Plus;
      A     "ВыбрСуп2";
      A     "ВыбрГор";
      );
      A     #Permission1;
      A     DB11.DBX 6.2;
      AN    "MSTT_1".B_Reset;
      =     DB34.DBX 4.7;
NETWORK
TITLE = Traversing key minus
      A(;
      O     "MSTT_1".B_Uminus;
      O;
      A     "КнАктВП";
      A     "HHU".S2_Minus;
      A     "ВыбрСуп2";
      A     "ВыбрГор";
      );
      A     #Permission1;
      A     DB11.DBX 6.2;
      AN    "MSTT_1".B_Reset;
      =     DB34.DBX 4.6;
NETWORK
TITLE = Delay reference point approach
      A     "БазоваяU";
      A     DB11.DBX 7.2;
      =     DB34.DBX 12.7;
NETWORK
TITLE = Activate fixed feed 1
      AN    "ПерАварВыклЛВС";
      =     DB34.DBX 3.2;
NETWORK
TITLE = Feed stop/spindle stop
      AN    #Permission1;
      AN    "РазрАвтонастр";
      =     DB34.DBX 4.3;
NETWORK
TITLE = Delete distance to go/Spindle-Reset
      A(;
      AN    #Permission1;
      A     DB11.DBX 6.2;
      O     "MSTT_1".B_Reset;
      );
      AN    "РазрАвтонастр";
      =     DB34.DBX 2.2;
NETWORK
TITLE = Hardware limit switch plus
      AN    "ОПW+";
      =     DB35.DBX 12.1;
NETWORK
TITLE = Hardware limit switch minus
      AN    "ОПW-";
      =     DB35.DBX 12.0;
NETWORK
TITLE = Controller enable
      A     DB35.DBX 93.5;
      A     "ТГотУЧПУ";
      =     L 4.0;
      A     L 4.0;
      BLD   102;
      =     DB35.DBX 2.1;
      A     L 4.0;
      BLD   102;
      =     DB35.DBX 21.7;
      A     L 4.0;
      BLD   102;
      =     Q 3.1;
      A     L 4.0;
      NOT;
      =     DB35.DBX 2.3;
NETWORK
TITLE = Traversing key plus
      A(;
      O     "MSTT_1".B_Wplus;
      O;
      A     "КнАктВП";
      A     "HHU".S3_Plus;
      A     "ВыбрСуп2";
      A     "ВыбрВерт";
      );
      A     #Permission2;
      A     DB11.DBX 6.2;
      AN    "MSTT_1".B_Reset;
      =     DB35.DBX 4.7;
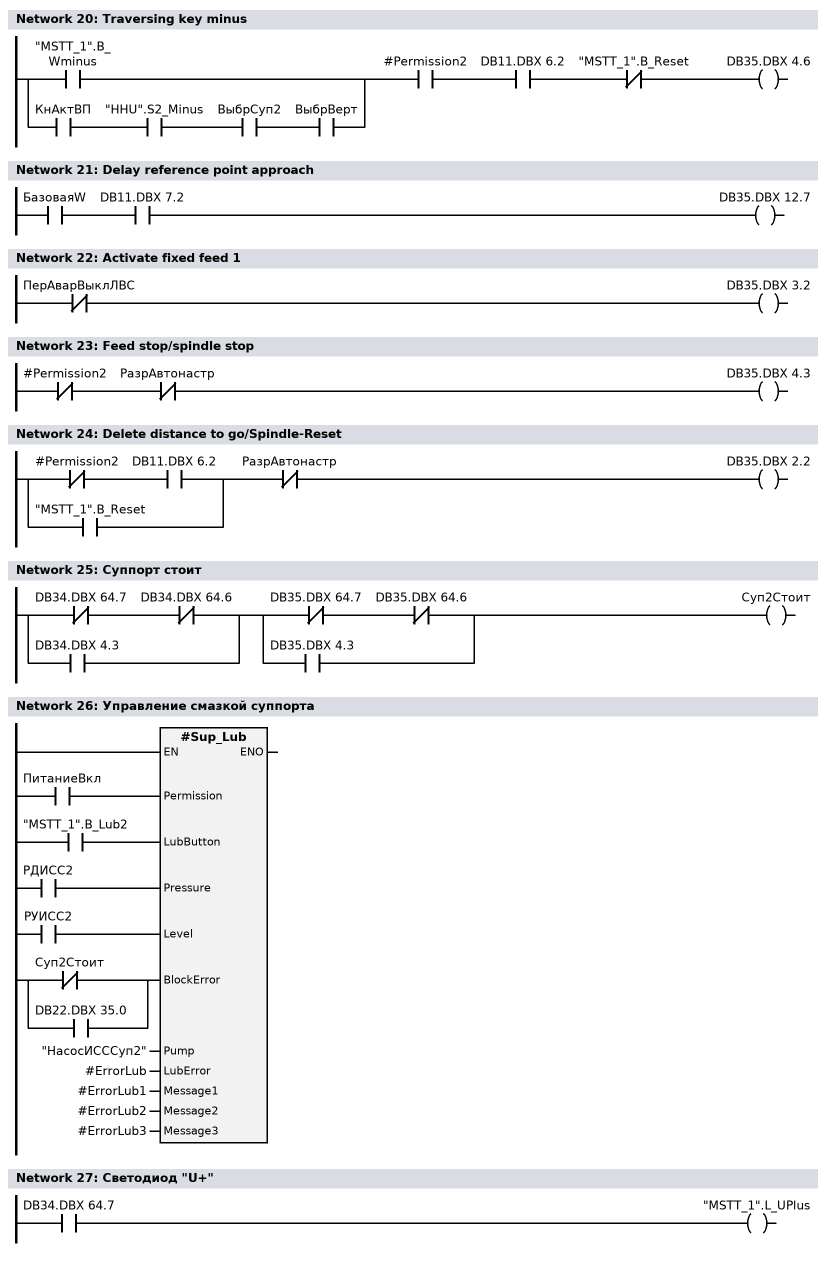
NETWORK
TITLE = Traversing key minus
      A(;
      O     "MSTT_1".B_Wminus;
      O;
      A     "КнАктВП";
      A     "HHU".S2_Minus;
      A     "ВыбрСуп2";
      A     "ВыбрВерт";
      );
      A     #Permission2;
      A     DB11.DBX 6.2;
      AN    "MSTT_1".B_Reset;
      =     DB35.DBX 4.6;
NETWORK
TITLE = Delay reference point approach
      A     "БазоваяW";
      A     DB11.DBX 7.2;
      =     DB35.DBX 12.7;
NETWORK
TITLE = Activate fixed feed 1
      AN    "ПерАварВыклЛВС";
      =     DB35.DBX 3.2;
NETWORK
TITLE = Feed stop/spindle stop
      AN    #Permission2;
      AN    "РазрАвтонастр";
      =     DB35.DBX 4.3;
NETWORK
TITLE = Delete distance to go/Spindle-Reset
      A(;
      AN    #Permission2;
      A     DB11.DBX 6.2;
      O     "MSTT_1".B_Reset;
      );
      AN    "РазрАвтонастр";
      =     DB35.DBX 2.2;
NETWORK
TITLE = Суппорт стоит
      A(;
      AN    DB34.DBX 64.7;
      AN    DB34.DBX 64.6;
      O     DB34.DBX 4.3;
      );
      A(;
      AN    DB35.DBX 64.7;
      AN    DB35.DBX 64.6;
      O     DB35.DBX 4.3;
      );
      =     "Суп2Стоит";
NETWORK
TITLE = Управление смазкой суппорта
      A     "ПитаниеВкл";
      =     L 4.0;
      BLD   103;
      A     "MSTT_1".B_Lub2;
      =     L 4.1;
      BLD   103;
      A     "РДИСС2";
      =     L 4.2;
      BLD   103;
      A     "РУИСС2";
      =     L 4.3;
      BLD   103;
      A(;
      ON    "Суп2Стоит";
      O     DB22.DBX 35.0;
      );
      =     L 4.4;
      BLD   103;
      CALL  #Sup_Lub (
           Permission               := L 4.0,
           LubButton                := L 4.1,
           Pressure                 := L 4.2,
           Level                    := L 4.3,
           BlockError               := L 4.4,
           Pump                     := "НасосИСССуп2",
           LubError                 := #ErrorLub,
           Message1                 := #ErrorLub1,
           Message2                 := #ErrorLub2,
           Message3                 := #ErrorLub3);
      NOP   0;
NETWORK
TITLE = Светодиод "U+"
      A     DB34.DBX 64.7;
      =     "MSTT_1".L_UPlus;
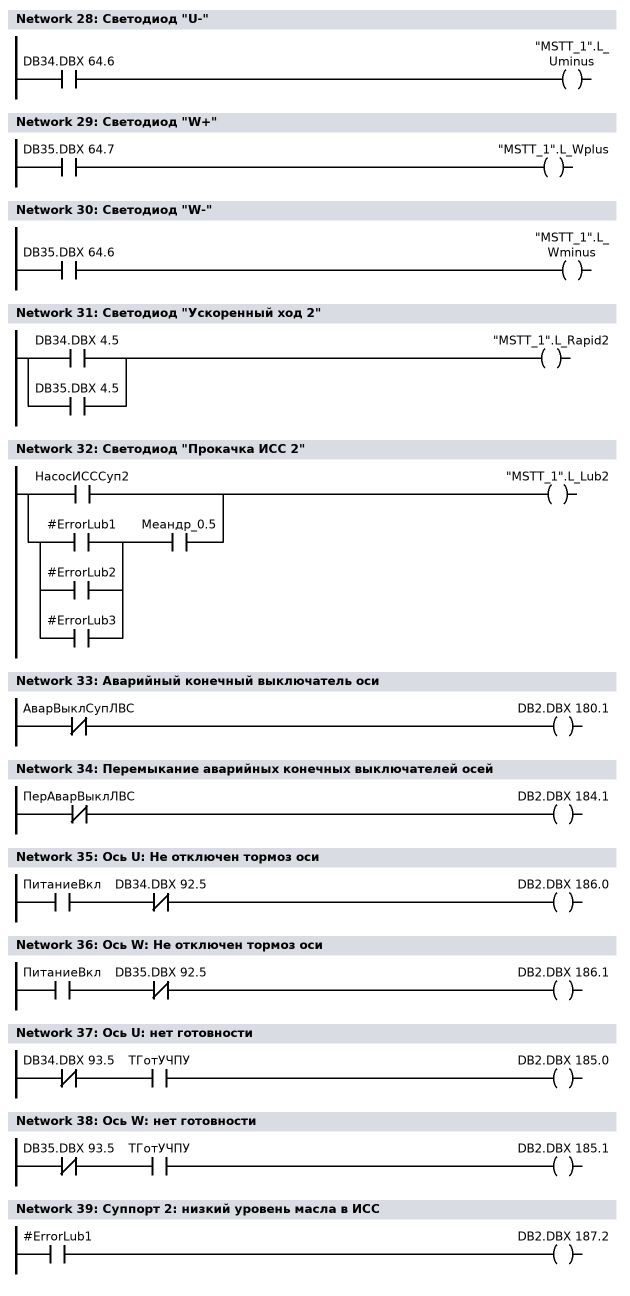
NETWORK
TITLE = Светодиод "U-"
      A     DB34.DBX 64.6;
      =     "MSTT_1".L_Uminus;
NETWORK
TITLE = Светодиод "W+"
      A     DB35.DBX 64.7;
      =     "MSTT_1".L_Wplus;
NETWORK
TITLE = Светодиод "W-"
      A     DB35.DBX 64.6;
      =     "MSTT_1".L_Wminus;
NETWORK
TITLE = Светодиод "Ускоренный ход 2"
      O     DB34.DBX 4.5;
      O     DB35.DBX 4.5;
      =     "MSTT_1".L_Rapid2;
NETWORK
TITLE = Светодиод "Прокачка ИСС 2"
      O     "НасосИСССуп2";
      O;
      A(;
      O     #ErrorLub1;
      O     #ErrorLub2;
      O     #ErrorLub3;
      );
      A     "Меандр_0.5";
      =     "MSTT_1".L_Lub2;
NETWORK
TITLE = Аварийный конечный выключатель оси
      AN    "АварВыклСупЛВС";
      =     DB2.DBX 180.1;
NETWORK
TITLE = Перемыкание аварийных конечных выключателей осей
      AN    "ПерАварВыклЛВС";
      =     DB2.DBX 184.1;
NETWORK
TITLE = Ось U: Не отключен тормоз оси
      A     "ПитаниеВкл";
      AN    DB34.DBX 92.5;
      =     DB2.DBX 186.0;
NETWORK
TITLE = Ось W: Не отключен тормоз оси
      A     "ПитаниеВкл";
      AN    DB35.DBX 92.5;
      =     DB2.DBX 186.1;
NETWORK
TITLE = Ось U: нет готовности
      AN    DB34.DBX 93.5;
      A     "ТГотУЧПУ";
      =     DB2.DBX 185.0;
NETWORK
TITLE = Ось W: нет готовности
      AN    DB35.DBX 93.5;
      A     "ТГотУЧПУ";
      =     DB2.DBX 185.1;
NETWORK
TITLE = Суппорт 2: низкий уровень масла в ИСС 
      A     #ErrorLub1;
      =     DB2.DBX 187.2;
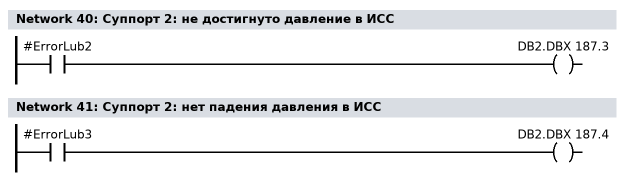
NETWORK
TITLE = Суппорт 2: не достигнуто давление в ИСС
      A     #ErrorLub2;
      =     DB2.DBX 187.3;
NETWORK
TITLE = Суппорт 2: нет падения давления в ИСС
      A     #ErrorLub3;
      =     DB2.DBX 187.4;
END_FUNCTION_BLOCK

FUNCTION_BLOCK "Support3_Ctrl"	// FB 103
AUTHOR : SEDIN
VERSION : 0.1
VAR
  Auxiliary : ARRAY  [0 .. 15 ] OF //Вспомогательная ячейка
  BOOL ;
  Unbrake1 : BOOL ;	//Требование разжима оси 1
  Unbrake2 : BOOL ;	//Требование разжима оси 2
  ErrorLub : BOOL ;	//Ошибка ИСС
  Sup_Lub : FB 121;	//Управление смазкой суппорта
  StartFC18_1 : BOOL ;	//Старт FC18
  StopFC18_1 : BOOL ;	//Остановка FC18
  InPosFC18_1 : BOOL ;	//Выполнение FC18
  ErrorFC18_1 : BOOL ;	//Ошибка FC18
  StartFC18_2 : BOOL ;	//Старт FC18
  StopFC18_2 : BOOL ;	//Остановка FC18
  InPosFC18_2 : BOOL ;	//Выполнение FC18
  ErrorFC18_2 : BOOL ;	//Ошибка FC18
  StateFC18_1 : BYTE ;	//Состояние FC18
  StateFC18_2 : BYTE ;	//Состояние FC18
END_VAR
VAR_TEMP
  Permission : BOOL ;	//Разрешение работы суппорта
  Permission1 : BOOL ;	//Разрешение работы суппорта, ось 1
  Permission2 : BOOL ;	//Разрешение работы суппорта, ось 2
  JogStop : BOOL ;	//Останов подачи в ручном режиме
  Stop1 : BOOL ;	//Суппорт стоит, ось 1
  Stop2 : BOOL ;	//Суппорт стоит, ось 2
  ErrorLub1 : BOOL ;	//Низкий уровень масла в ИСС
  ErrorLub2 : BOOL ;	//Не достигнуто давление в ИСС
  ErrorLub3 : BOOL ;	//Нет падения давления в ИСС
  GAct : INT ;	//Текущая G-функция 15 группы
END_VAR
BEGIN
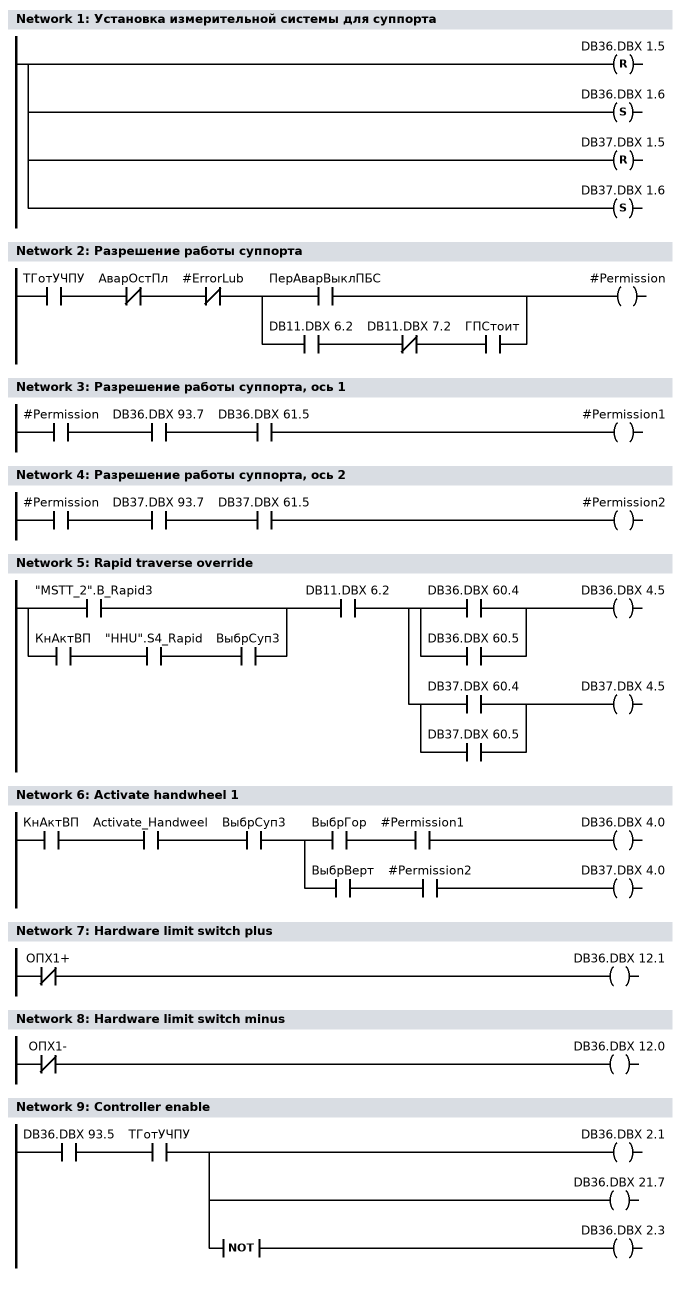
NETWORK
TITLE = Установка измерительной системы для суппорта
      SET;
      R     DB36.DBX 1.5;
      S     DB36.DBX 1.6;
      R     DB37.DBX 1.5;
      S     DB37.DBX 1.6;
NETWORK
TITLE = Разрешение работы суппорта
      A     "ТГотУЧПУ";
      AN    "АварОстПл";
      AN    #ErrorLub;
      A(;
      O     "ПерАварВыклПБС";
      O;
      A     DB11.DBX 6.2;
      AN    DB11.DBX 7.2;
      A     "ГПСтоит";
      );
      =     #Permission;
NETWORK
TITLE = Разрешение работы суппорта, ось 1
      A     #Permission;
      A     DB36.DBX 93.7;
      A     DB36.DBX 61.5;
      =     #Permission1;
NETWORK
TITLE = Разрешение работы суппорта, ось 2
      A     #Permission;
      A     DB37.DBX 93.7;
      A     DB37.DBX 61.5;
      =     #Permission2;
NETWORK
TITLE = Rapid traverse override
      A(;
      O     "MSTT_2".B_Rapid3;
      O;
      A     "КнАктВП";
      A     "HHU".S4_Rapid;
      A     "ВыбрСуп3";
      );
      A     DB11.DBX 6.2;
      =     L 4.0;
      A     L 4.0;
      A(;
      O     DB36.DBX 60.4;
      O     DB36.DBX 60.5;
      );
      =     DB36.DBX 4.5;
      A     L 4.0;
      A(;
      O     DB37.DBX 60.4;
      O     DB37.DBX 60.5;
      );
      =     DB37.DBX 4.5;
NETWORK
TITLE = Activate handwheel 1
      A     "КнАктВП";
      A     "Activate_Handweel";
      A     "ВыбрСуп3";
      =     L 4.0;
      A     L 4.0;
      A     "ВыбрГор";
      A     #Permission1;
      =     DB36.DBX 4.0;
      A     L 4.0;
      A     "ВыбрВерт";
      A     #Permission2;
      =     DB37.DBX 4.0;
NETWORK
TITLE = Hardware limit switch plus
      AN    "ОПX1+";
      =     DB36.DBX 12.1;
NETWORK
TITLE = Hardware limit switch minus
      AN    "ОПX1-";
      =     DB36.DBX 12.0;
NETWORK
TITLE = Controller enable
      A     DB36.DBX 93.5;
      A     "ТГотУЧПУ";
      =     L 4.0;
      A     L 4.0;
      BLD   102;
      =     DB36.DBX 2.1;
      A     L 4.0;
      BLD   102;
      =     DB36.DBX 21.7;
      A     L 4.0;
      NOT;
      =     DB36.DBX 2.3;
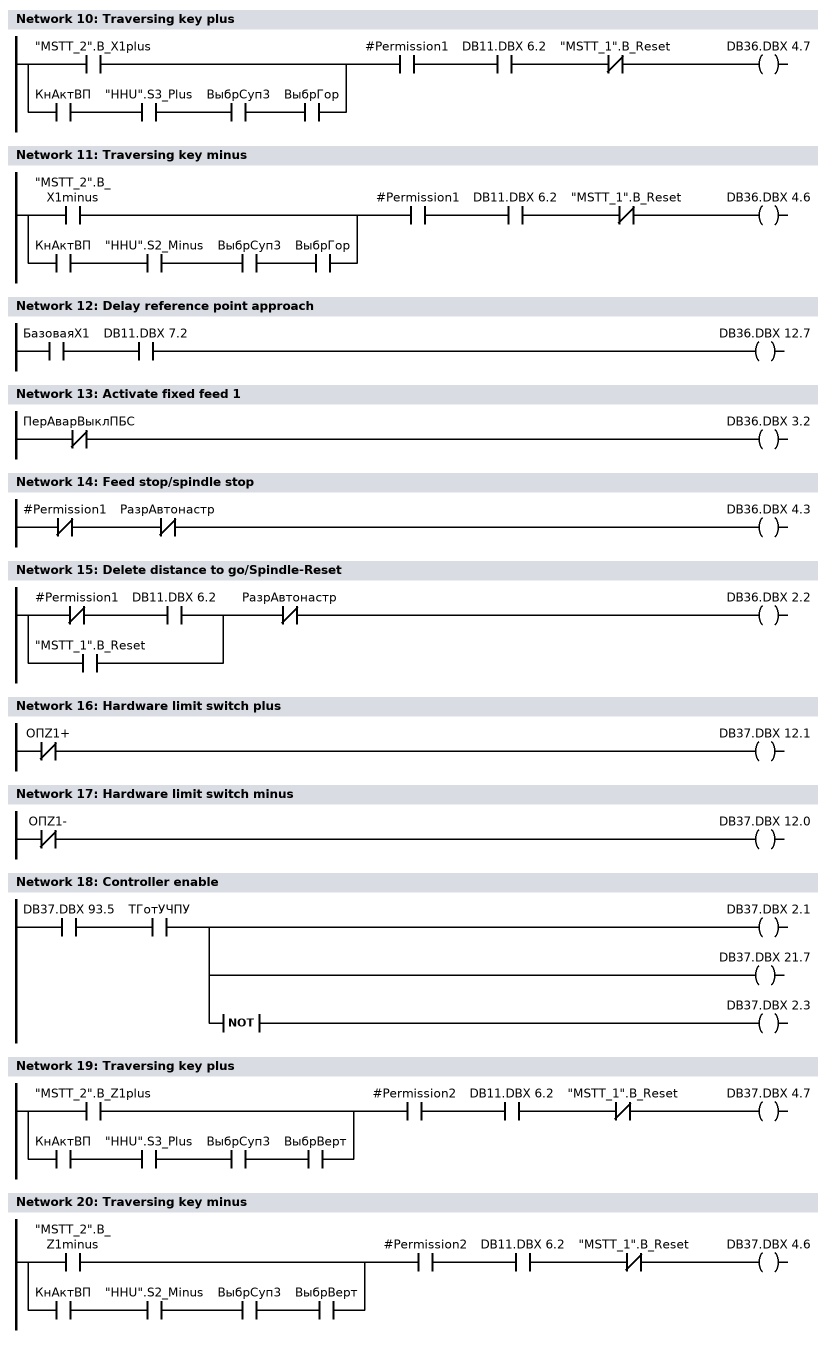
NETWORK
TITLE = Traversing key plus
      A(;
      O     "MSTT_2".B_X1plus;
      O;
      A     "КнАктВП";
      A     "HHU".S3_Plus;
      A     "ВыбрСуп3";
      A     "ВыбрГор";
      );
      A     #Permission1;
      A     DB11.DBX 6.2;
      AN    "MSTT_1".B_Reset;
      =     DB36.DBX 4.7;
NETWORK
TITLE = Traversing key minus
      A(;
      O     "MSTT_2".B_X1minus;
      O;
      A     "КнАктВП";
      A     "HHU".S2_Minus;
      A     "ВыбрСуп3";
      A     "ВыбрГор";
      );
      A     #Permission1;
      A     DB11.DBX 6.2;
      AN    "MSTT_1".B_Reset;
      =     DB36.DBX 4.6;
NETWORK
TITLE = Delay reference point approach
      A     "БазоваяX1";
      A     DB11.DBX 7.2;
      =     DB36.DBX 12.7;
NETWORK
TITLE = Activate fixed feed 1
      AN    "ПерАварВыклПБС";
      =     DB36.DBX 3.2;
NETWORK
TITLE = Feed stop/spindle stop
      AN    #Permission1;
      AN    "РазрАвтонастр";
      =     DB36.DBX 4.3;
NETWORK
TITLE = Delete distance to go/Spindle-Reset
      A(;
      AN    #Permission1;
      A     DB11.DBX 6.2;
      O     "MSTT_1".B_Reset;
      );
      AN    "РазрАвтонастр";
      =     DB36.DBX 2.2;
NETWORK
TITLE = Hardware limit switch plus
      AN    "ОПZ1+";
      =     DB37.DBX 12.1;
NETWORK
TITLE = Hardware limit switch minus
      AN    "ОПZ1-";
      =     DB37.DBX 12.0;
NETWORK
TITLE = Controller enable
      A     DB37.DBX 93.5;
      A     "ТГотУЧПУ";
      =     L 4.0;
      A     L 4.0;
      BLD   102;
      =     DB37.DBX 2.1;
      A     L 4.0;
      BLD   102;
      =     DB37.DBX 21.7;
      A     L 4.0;
      NOT;
      =     DB37.DBX 2.3;
NETWORK
TITLE = Traversing key plus
      A(;
      O     "MSTT_2".B_Z1plus;
      O;
      A     "КнАктВП";
      A     "HHU".S3_Plus;
      A     "ВыбрСуп3";
      A     "ВыбрВерт";
      );
      A     #Permission2;
      A     DB11.DBX 6.2;
      AN    "MSTT_1".B_Reset;
      =     DB37.DBX 4.7;
NETWORK
TITLE = Traversing key minus
      A(;
      O     "MSTT_2".B_Z1minus;
      O;
      A     "КнАктВП";
      A     "HHU".S2_Minus;
      A     "ВыбрСуп3";
      A     "ВыбрВерт";
      );
      A     #Permission2;
      A     DB11.DBX 6.2;
      AN    "MSTT_1".B_Reset;
      =     DB37.DBX 4.6;
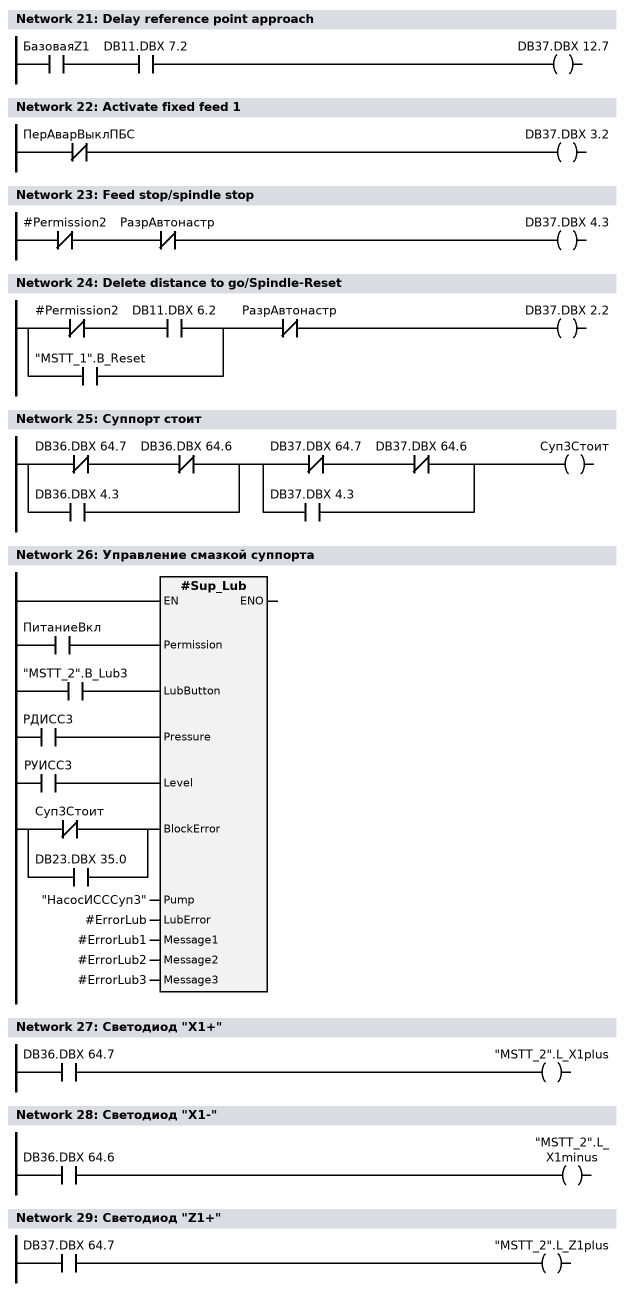
NETWORK
TITLE = Delay reference point approach
      A     "БазоваяZ1";
      A     DB11.DBX 7.2;
      =     DB37.DBX 12.7;
NETWORK
TITLE = Activate fixed feed 1
      AN    "ПерАварВыклПБС";
      =     DB37.DBX 3.2;
NETWORK
TITLE = Feed stop/spindle stop
      AN    #Permission2;
      AN    "РазрАвтонастр";
      =     DB37.DBX 4.3;
NETWORK
TITLE = Delete distance to go/Spindle-Reset
      A(;
      AN    #Permission2;
      A     DB11.DBX 6.2;
      O     "MSTT_1".B_Reset;
      );
      AN    "РазрАвтонастр";
      =     DB37.DBX 2.2;
NETWORK
TITLE = Суппорт стоит
      A(;
      AN    DB36.DBX 64.7;
      AN    DB36.DBX 64.6;
      O     DB36.DBX 4.3;
      );
      A(;
      AN    DB37.DBX 64.7;
      AN    DB37.DBX 64.6;
      O     DB37.DBX 4.3;
      );
      =     "Суп3Стоит";
NETWORK
TITLE = Управление смазкой суппорта
      A     "ПитаниеВкл";
      =     L 4.0;
      BLD   103;
      A     "MSTT_2".B_Lub3;
      =     L 4.1;
      BLD   103;
      A     "РДИСС3";
      =     L 4.2;
      BLD   103;
      A     "РУИСС3";
      =     L 4.3;
      BLD   103;
      A(;
      ON    "Суп3Стоит";
      O     DB23.DBX 35.0;
      );
      =     L 4.4;
      BLD   103;
      CALL  #Sup_Lub (
           Permission               := L 4.0,
           LubButton                := L 4.1,
           Pressure                 := L 4.2,
           Level                    := L 4.3,
           BlockError               := L 4.4,
           Pump                     := "НасосИСССуп3",
           LubError                 := #ErrorLub,
           Message1                 := #ErrorLub1,
           Message2                 := #ErrorLub2,
           Message3                 := #ErrorLub3);
      NOP   0;
NETWORK
TITLE = Светодиод "X1+"
      A     DB36.DBX 64.7;
      =     "MSTT_2".L_X1plus;
NETWORK
TITLE = Светодиод "X1-"
      A     DB36.DBX 64.6;
      =     "MSTT_2".L_X1minus;
NETWORK
TITLE = Светодиод "Z1+"
      A     DB37.DBX 64.7;
      =     "MSTT_2".L_Z1plus;
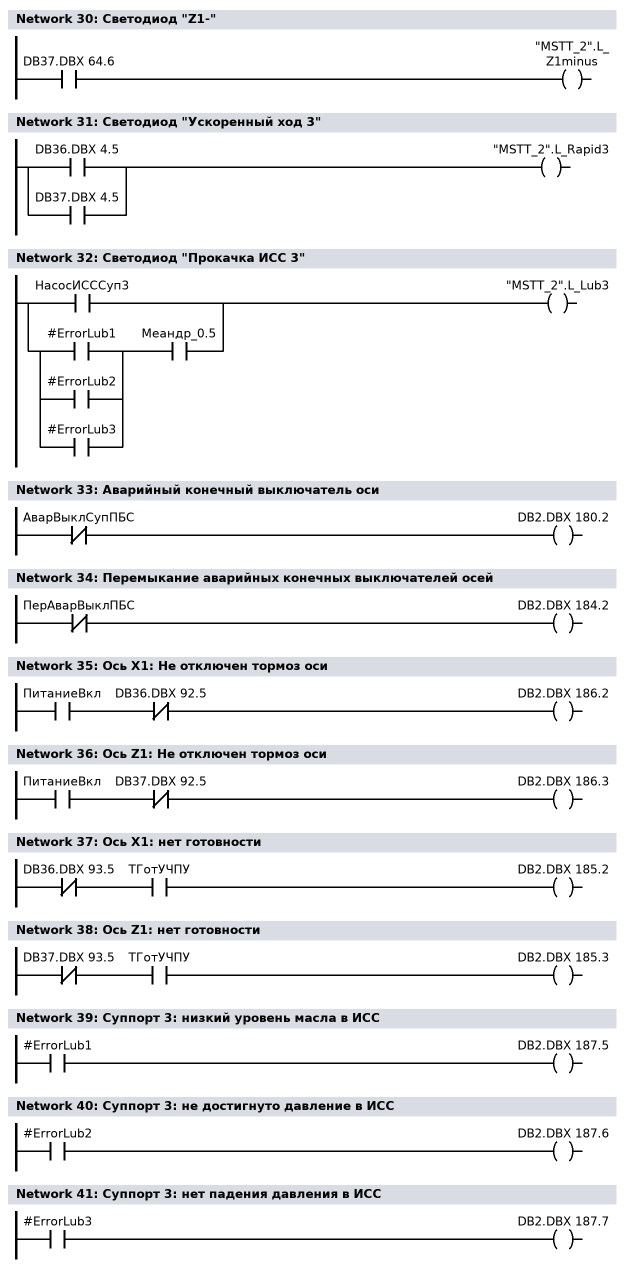
NETWORK
TITLE = Светодиод "Z1-"
      A     DB37.DBX 64.6;
      =     "MSTT_2".L_Z1minus;
NETWORK
TITLE = Светодиод "Ускоренный ход 3"
      O     DB36.DBX 4.5;
      O     DB37.DBX 4.5;
      =     "MSTT_2".L_Rapid3;
NETWORK
TITLE = Светодиод "Прокачка ИСС 3"
      O     "НасосИСССуп3";
      O;
      A(;
      O     #ErrorLub1;
      O     #ErrorLub2;
      O     #ErrorLub3;
      );
      A     "Меандр_0.5";
      =     "MSTT_2".L_Lub3;
NETWORK
TITLE = Аварийный конечный выключатель оси
      AN    "АварВыклСупПБС";
      =     DB2.DBX 180.2;
NETWORK
TITLE = Перемыкание аварийных конечных выключателей осей
      AN    "ПерАварВыклПБС";
      =     DB2.DBX 184.2;
NETWORK
TITLE = Ось X1: Не отключен тормоз оси
      A     "ПитаниеВкл";
      AN    DB36.DBX 92.5;
      =     DB2.DBX 186.2;
NETWORK
TITLE = Ось Z1: Не отключен тормоз оси
      A     "ПитаниеВкл";
      AN    DB37.DBX 92.5;
      =     DB2.DBX 186.3;
NETWORK
TITLE = Ось X1: нет готовности
      AN    DB36.DBX 93.5;
      A     "ТГотУЧПУ";
      =     DB2.DBX 185.2;
NETWORK
TITLE = Ось Z1: нет готовности
      AN    DB37.DBX 93.5;
      A     "ТГотУЧПУ";
      =     DB2.DBX 185.3;
NETWORK
TITLE = Суппорт 3: низкий уровень масла в ИСС 
      A     #ErrorLub1;
      =     DB2.DBX 187.5;
NETWORK
TITLE = Суппорт 3: не достигнуто давление в ИСС
      A     #ErrorLub2;
      =     DB2.DBX 187.6;
NETWORK
TITLE = Суппорт 3: нет падения давления в ИСС
      A     #ErrorLub3;
      =     DB2.DBX 187.7;
END_FUNCTION_BLOCK

FUNCTION_BLOCK "Support4_Ctrl"	// FB 104
AUTHOR : SEDIN
VERSION : 0.1
VAR
  Auxiliary : ARRAY  [0 .. 15 ] OF //Вспомогательная ячейка
  BOOL ;
  Unbrake1 : BOOL ;	//Требование разжима оси 1
  Unbrake2 : BOOL ;	//Требование разжима оси 2
  ErrorLub : BOOL ;	//Ошибка ИСС
  Sup_Lub : FB 121;	//Управление смазкой суппорта
  StartFC18_1 : BOOL ;	//Старт FC18
  StopFC18_1 : BOOL ;	//Остановка FC18
  InPosFC18_1 : BOOL ;	//Выполнение FC18
  ErrorFC18_1 : BOOL ;	//Ошибка FC18
  StartFC18_2 : BOOL ;	//Старт FC18
  StopFC18_2 : BOOL ;	//Остановка FC18
  InPosFC18_2 : BOOL ;	//Выполнение FC18
  ErrorFC18_2 : BOOL ;	//Ошибка FC18
  StateFC18_1 : BYTE ;	//Состояние FC18
  StateFC18_2 : BYTE ;	//Состояние FC18
END_VAR
VAR_TEMP
  Permission : BOOL ;	//Разрешение работы суппорта
  Permission1 : BOOL ;	//Разрешение работы суппорта, ось 1
  Permission2 : BOOL ;	//Разрешение работы суппорта, ось 2
  JogStop : BOOL ;	//Останов подачи в ручном режиме
  Stop1 : BOOL ;	//Суппорт стоит, ось 1
  Stop2 : BOOL ;	//Суппорт стоит, ось 2
  ErrorLub1 : BOOL ;	//Низкий уровень масла в ИСС
  ErrorLub2 : BOOL ;	//Не достигнуто давление в ИСС
  ErrorLub3 : BOOL ;	//Нет падения давления в ИСС
  GAct : INT ;	//Текущая G-функция 15 группы
END_VAR
BEGIN
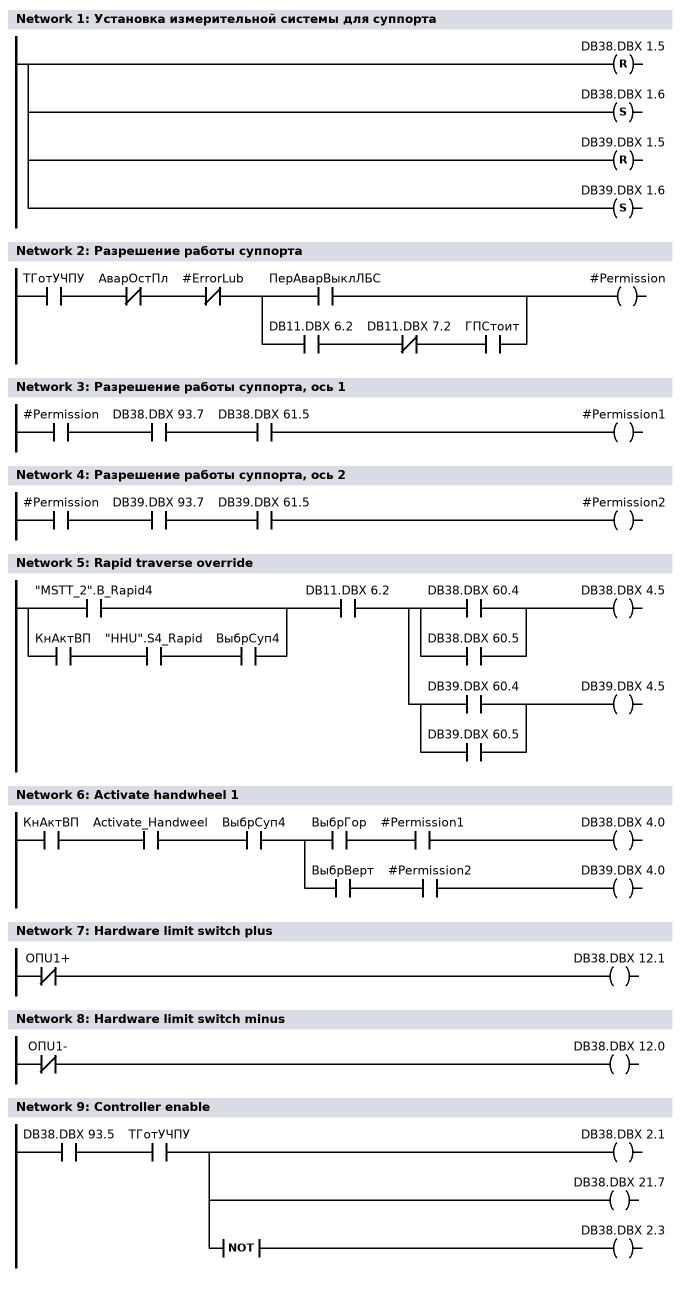
NETWORK
TITLE = Установка измерительной системы для суппорта
      SET;
      R     DB38.DBX 1.5;
      S     DB38.DBX 1.6;
      R     DB39.DBX 1.5;
      S     DB39.DBX 1.6;
NETWORK
TITLE = Разрешение работы суппорта
      A     "ТГотУЧПУ";
      AN    "АварОстПл";
      AN    #ErrorLub;
      A(;
      O     "ПерАварВыклЛБС";
      O;
      A     DB11.DBX 6.2;
      AN    DB11.DBX 7.2;
      A     "ГПСтоит";
      );
      =     #Permission;
NETWORK
TITLE = Разрешение работы суппорта, ось 1
      A     #Permission;
      A     DB38.DBX 93.7;
      A     DB38.DBX 61.5;
      =     #Permission1;
NETWORK
TITLE = Разрешение работы суппорта, ось 2
      A     #Permission;
      A     DB39.DBX 93.7;
      A     DB39.DBX 61.5;
      =     #Permission2;
NETWORK
TITLE = Rapid traverse override
      A(;
      O     "MSTT_2".B_Rapid4;
      O;
      A     "КнАктВП";
      A     "HHU".S4_Rapid;
      A     "ВыбрСуп4";
      );
      A     DB11.DBX 6.2;
      =     L 4.0;
      A     L 4.0;
      A(;
      O     DB38.DBX 60.4;
      O     DB38.DBX 60.5;
      );
      =     DB38.DBX 4.5;
      A     L 4.0;
      A(;
      O     DB39.DBX 60.4;
      O     DB39.DBX 60.5;
      );
      =     DB39.DBX 4.5;
NETWORK
TITLE = Activate handwheel 1
      A     "КнАктВП";
      A     "Activate_Handweel";
      A     "ВыбрСуп4";
      =     L 4.0;
      A     L 4.0;
      A     "ВыбрГор";
      A     #Permission1;
      =     DB38.DBX 4.0;
      A     L 4.0;
      A     "ВыбрВерт";
      A     #Permission2;
      =     DB39.DBX 4.0;
NETWORK
TITLE = Hardware limit switch plus
      AN    "ОПU1+";
      =     DB38.DBX 12.1;
NETWORK
TITLE = Hardware limit switch minus
      AN    "ОПU1-";
      =     DB38.DBX 12.0;
NETWORK
TITLE = Controller enable
      A     DB38.DBX 93.5;
      A     "ТГотУЧПУ";
      =     L 4.0;
      A     L 4.0;
      BLD   102;
      =     DB38.DBX 2.1;
      A     L 4.0;
      BLD   102;
      =     DB38.DBX 21.7;
      A     L 4.0;
      NOT;
      =     DB38.DBX 2.3;
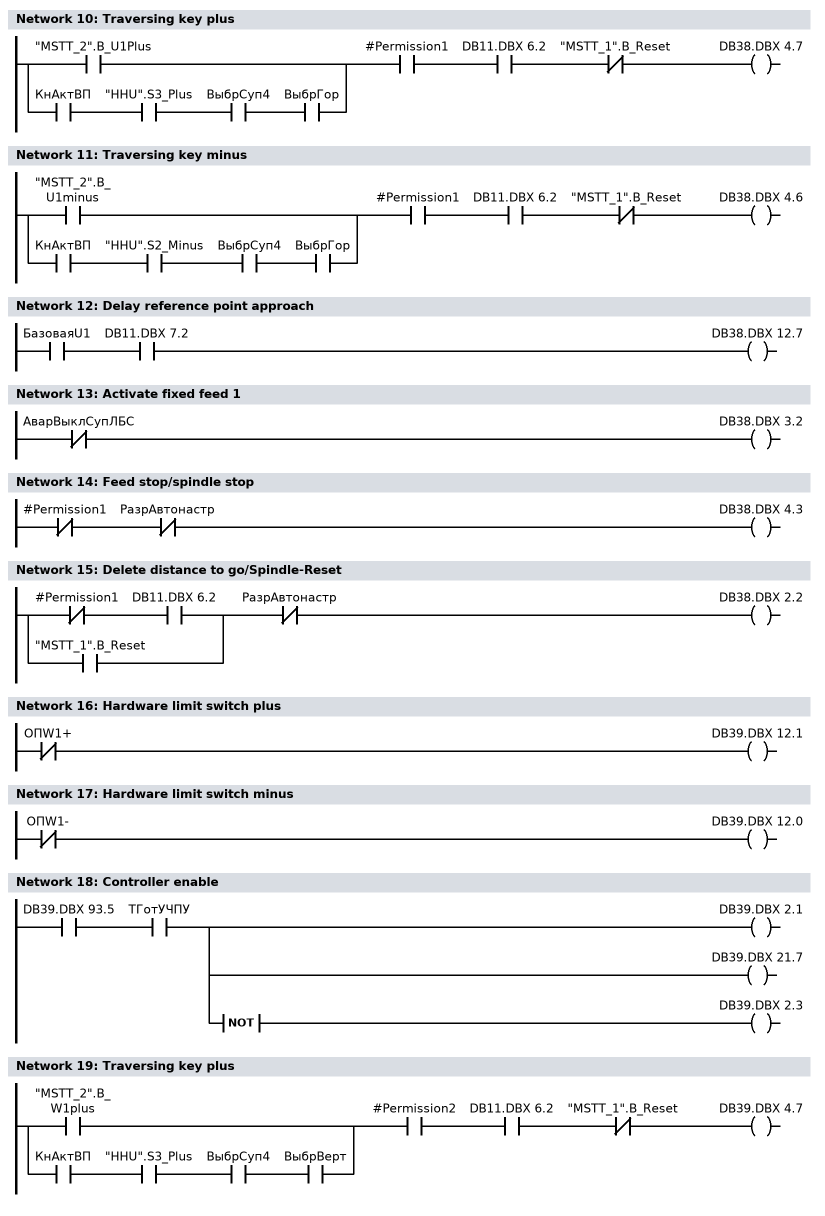
NETWORK
TITLE = Traversing key plus
      A(;
      O     "MSTT_2".B_U1Plus;
      O;
      A     "КнАктВП";
      A     "HHU".S3_Plus;
      A     "ВыбрСуп4";
      A     "ВыбрГор";
      );
      A     #Permission1;
      A     DB11.DBX 6.2;
      AN    "MSTT_1".B_Reset;
      =     DB38.DBX 4.7;
NETWORK
TITLE = Traversing key minus
      A(;
      O     "MSTT_2".B_U1minus;
      O;
      A     "КнАктВП";
      A     "HHU".S2_Minus;
      A     "ВыбрСуп4";
      A     "ВыбрГор";
      );
      A     #Permission1;
      A     DB11.DBX 6.2;
      AN    "MSTT_1".B_Reset;
      =     DB38.DBX 4.6;
NETWORK
TITLE = Delay reference point approach
      A     "БазоваяU1";
      A     DB11.DBX 7.2;
      =     DB38.DBX 12.7;
NETWORK
TITLE = Activate fixed feed 1
      AN    "АварВыклСупЛБС";
      =     DB38.DBX 3.2;
NETWORK
TITLE = Feed stop/spindle stop
      AN    #Permission1;
      AN    "РазрАвтонастр";
      =     DB38.DBX 4.3;
NETWORK
TITLE = Delete distance to go/Spindle-Reset
      A(;
      AN    #Permission1;
      A     DB11.DBX 6.2;
      O     "MSTT_1".B_Reset;
      );
      AN    "РазрАвтонастр";
      =     DB38.DBX 2.2;
NETWORK
TITLE = Hardware limit switch plus
      AN    "ОПW1+";
      =     DB39.DBX 12.1;
NETWORK
TITLE = Hardware limit switch minus
      AN    "ОПW1-";
      =     DB39.DBX 12.0;
NETWORK
TITLE = Controller enable
      A     DB39.DBX 93.5;
      A     "ТГотУЧПУ";
      =     L 4.0;
      A     L 4.0;
      BLD   102;
      =     DB39.DBX 2.1;
      A     L 4.0;
      BLD   102;
      =     DB39.DBX 21.7;
      A     L 4.0;
      NOT;
      =     DB39.DBX 2.3;
NETWORK
TITLE = Traversing key plus
      A(;
      O     "MSTT_2".B_W1plus;
      O;
      A     "КнАктВП";
      A     "HHU".S3_Plus;
      A     "ВыбрСуп4";
      A     "ВыбрВерт";
      );
      A     #Permission2;
      A     DB11.DBX 6.2;
      AN    "MSTT_1".B_Reset;
      =     DB39.DBX 4.7;
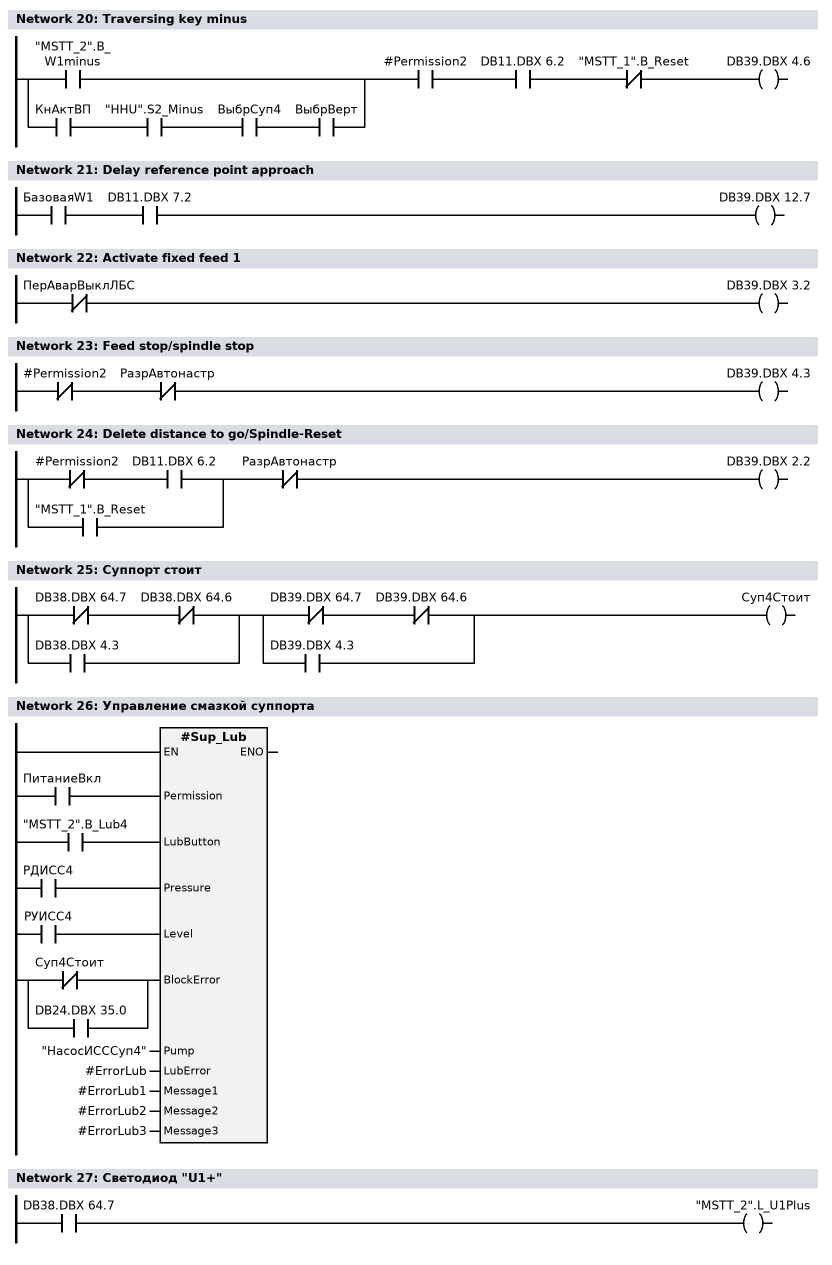
NETWORK
TITLE = Traversing key minus
      A(;
      O     "MSTT_2".B_W1minus;
      O;
      A     "КнАктВП";
      A     "HHU".S2_Minus;
      A     "ВыбрСуп4";
      A     "ВыбрВерт";
      );
      A     #Permission2;
      A     DB11.DBX 6.2;
      AN    "MSTT_1".B_Reset;
      =     DB39.DBX 4.6;
NETWORK
TITLE = Delay reference point approach
      A     "БазоваяW1";
      A     DB11.DBX 7.2;
      =     DB39.DBX 12.7;
NETWORK
TITLE = Activate fixed feed 1
      AN    "ПерАварВыклЛБС";
      =     DB39.DBX 3.2;
NETWORK
TITLE = Feed stop/spindle stop
      AN    #Permission2;
      AN    "РазрАвтонастр";
      =     DB39.DBX 4.3;
NETWORK
TITLE = Delete distance to go/Spindle-Reset
      A(;
      AN    #Permission2;
      A     DB11.DBX 6.2;
      O     "MSTT_1".B_Reset;
      );
      AN    "РазрАвтонастр";
      =     DB39.DBX 2.2;
NETWORK
TITLE = Суппорт стоит
      A(;
      AN    DB38.DBX 64.7;
      AN    DB38.DBX 64.6;
      O     DB38.DBX 4.3;
      );
      A(;
      AN    DB39.DBX 64.7;
      AN    DB39.DBX 64.6;
      O     DB39.DBX 4.3;
      );
      =     "Суп4Стоит";
NETWORK
TITLE = Управление смазкой суппорта
      A     "ПитаниеВкл";
      =     L 4.0;
      BLD   103;
      A     "MSTT_2".B_Lub4;
      =     L 4.1;
      BLD   103;
      A     "РДИСС4";
      =     L 4.2;
      BLD   103;
      A     "РУИСС4";
      =     L 4.3;
      BLD   103;
      A(;
      ON    "Суп4Стоит";
      O     DB24.DBX 35.0;
      );
      =     L 4.4;
      BLD   103;
      CALL  #Sup_Lub (
           Permission               := L 4.0,
           LubButton                := L 4.1,
           Pressure                 := L 4.2,
           Level                    := L 4.3,
           BlockError               := L 4.4,
           Pump                     := "НасосИСССуп4",
           LubError                 := #ErrorLub,
           Message1                 := #ErrorLub1,
           Message2                 := #ErrorLub2,
           Message3                 := #ErrorLub3);
      NOP   0;
NETWORK
TITLE = Светодиод "U1+"
      A     DB38.DBX 64.7;
      =     "MSTT_2".L_U1Plus;
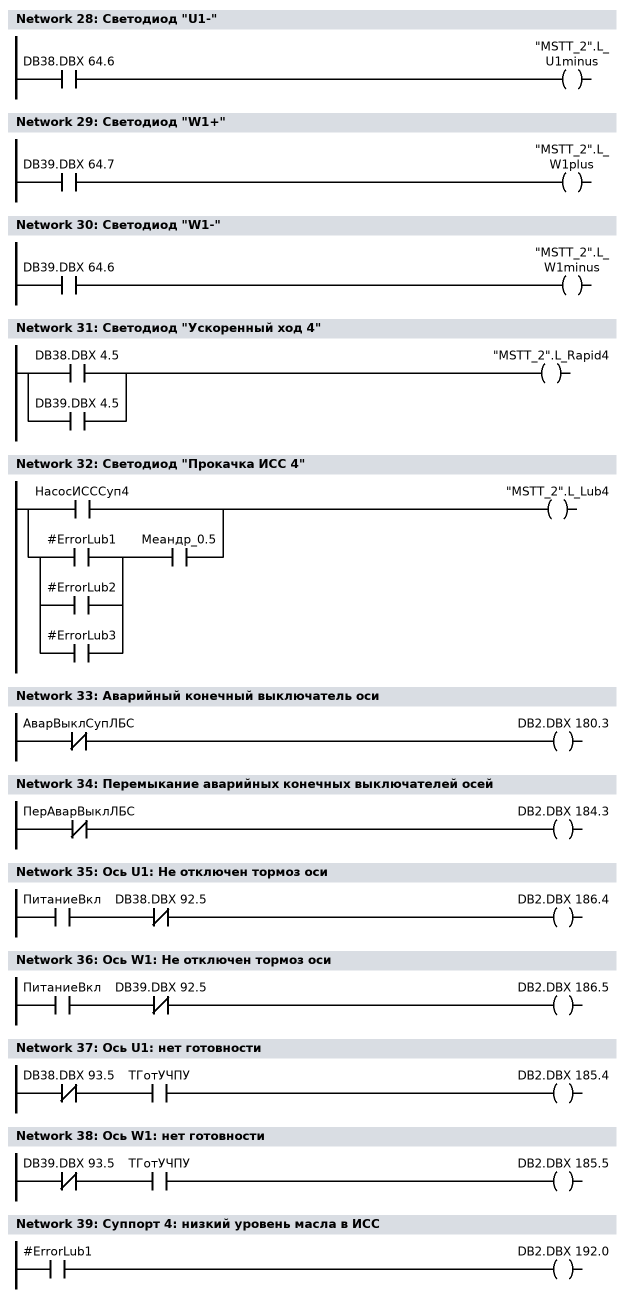
NETWORK
TITLE = Светодиод "U1-"
      A     DB38.DBX 64.6;
      =     "MSTT_2".L_U1minus;
NETWORK
TITLE = Светодиод "W1+"
      A     DB39.DBX 64.7;
      =     "MSTT_2".L_W1plus;
NETWORK
TITLE = Светодиод "W1-"
      A     DB39.DBX 64.6;
      =     "MSTT_2".L_W1minus;
NETWORK
TITLE = Светодиод "Ускоренный ход 4"
      O     DB38.DBX 4.5;
      O     DB39.DBX 4.5;
      =     "MSTT_2".L_Rapid4;
NETWORK
TITLE = Светодиод "Прокачка ИСС 4"
      O     "НасосИСССуп4";
      O;
      A(;
      O     #ErrorLub1;
      O     #ErrorLub2;
      O     #ErrorLub3;
      );
      A     "Меандр_0.5";
      =     "MSTT_2".L_Lub4;
NETWORK
TITLE = Аварийный конечный выключатель оси
      AN    "АварВыклСупЛБС";
      =     DB2.DBX 180.3;
NETWORK
TITLE = Перемыкание аварийных конечных выключателей осей
      AN    "ПерАварВыклЛБС";
      =     DB2.DBX 184.3;
NETWORK
TITLE = Ось U1: Не отключен тормоз оси
      A     "ПитаниеВкл";
      AN    DB38.DBX 92.5;
      =     DB2.DBX 186.4;
NETWORK
TITLE = Ось W1: Не отключен тормоз оси
      A     "ПитаниеВкл";
      AN    DB39.DBX 92.5;
      =     DB2.DBX 186.5;
NETWORK
TITLE = Ось U1: нет готовности
      AN    DB38.DBX 93.5;
      A     "ТГотУЧПУ";
      =     DB2.DBX 185.4;
NETWORK
TITLE = Ось W1: нет готовности
      AN    DB39.DBX 93.5;
      A     "ТГотУЧПУ";
      =     DB2.DBX 185.5;
NETWORK
TITLE = Суппорт 4: низкий уровень масла в ИСС 
      A     #ErrorLub1;
      =     DB2.DBX 192.0;
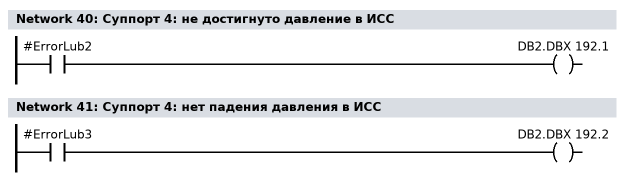
NETWORK
TITLE = Суппорт 4: не достигнуто давление в ИСС
      A     #ErrorLub2;
      =     DB2.DBX 192.1;
NETWORK
TITLE = Суппорт 4: нет падения давления в ИСС
      A     #ErrorLub3;
      =     DB2.DBX 192.2;
END_FUNCTION_BLOCK

FUNCTION_BLOCK "Lathe_Modes"	// FB 105
AUTHOR : SEDIN
VERSION : 0.1
VAR
  Auxiliary : ARRAY  [0 .. 15 ] OF //Вспомогательная ячейка
  BOOL ;
  Canal_1 : FB 106;
  Canal_2 : FB 107;
  Canal_3 : FB 108;
  Canal_4 : FB 109;
  Get_Pos : FB 2;
  Get_Rel1 : FB 2;
  Get_Rel2 : FB 2;
  Get_Rel3 : FB 2;
  Get_Rel4 : FB 2;
  NDR1 : BOOL ;	//Выполнение считывания блока FB2
  Err1 : BOOL ;	//Ошибка работы блока FB2
  NDR2 : BOOL ;	//Выполнение считывания блока FB2
  Err2 : BOOL ;	//Ошибка работы блока FB2
  NDR3 : BOOL ;	//Выполнение считывания блока FB2
  Err3 : BOOL ;	//Ошибка работы блока FB2
  NDR4 : BOOL ;	//Выполнение считывания блока FB2
  Err4 : BOOL ;	//Ошибка работы блока FB2
  NDR5 : BOOL ;	//Выполнение считывания блока FB2
  Err5 : BOOL ;	//Ошибка работы блока FB2
END_VAR
VAR_TEMP
  Ret1 : WORD ;	//Результат работы блока FB2
  Ret2 : WORD ;	//Результат работы блока FB2
  Ret3 : WORD ;	//Результат работы блока FB2
  Ret4 : WORD ;	//Результат работы блока FB2
  Ret5 : WORD ;	//Результат работы блока FB2
  NumChan : INT ;	//Номер канала
END_VAR
BEGIN
